(* Logix 5000 project; controller RSL5k_18_Template_noLib Emulate 5570 rev 32.11; software revision 32.02; part 6 of 16 *)
(* tags used below, declared in another part *)
   P_Intlk : BOOL;   // Unique Parameter Name for auto - discovery
(* P_Intlk, continued *)

ROUTINE Prescan   (* ladder *)
// Clear "lurking" Commands
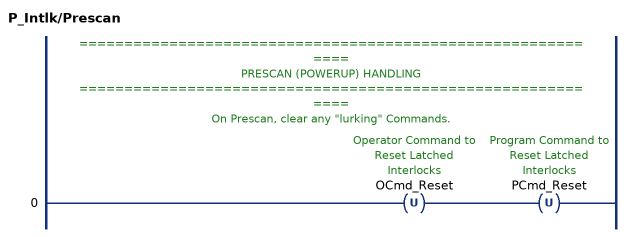
   // ============================================================
   // PRESCAN (POWERUP) HANDLING
   // ============================================================
   // On Prescan, clear any "lurking" Commands.
   0: OTU(OCmd_Reset)OTU(PCmd_Reset);
END_ROUTINE
END_ADD_ON_INSTRUCTION

ADD_ON_INSTRUCTION P_Perm   (* revision 4.10 .00 Release, vendor Rockwell Automation, ExecuteEnableInFalse *)
// Permissives
// Revision note:
// See Instruction Help for a summary of changes, and see 4.10 Release Notes for details.
// Help:
// Copyright © Rockwell Automation, Inc.  All Rights Reserved.
// This Instruction monitors up to 16 Permissive conditions.  It provides these features:
// *  The "OK" state of each Permissive Input is configurable.  By default,
//     each Input is 1 when OK to start, 0 when not OK to start.
// *  Permissives may be configured as Bypassable.  A separate Sts_NBPermOK
//     (Non-Bypassable Permissives OK) status is provided, which the destination
//     object can use for Bypass, Maintenance and other functions,
//     where Bypassable Permissives can be ignored.
// All Permissive Inputs must be in their configured "OK" states
// for the P_Perm instruction to provide a "PermOK" status.
// All non-bypassable Permissive inputs must be in their configured "OK" states
// for the P_Perm instruction to provide a "NBPermOK" status.
// For each Permissive condition, a Tag may be defined for navigation. Clicking
// the Permissive description will call up the associated Tag's Faceplate.
// SUMMARY OF CHANGES FROM PREVIOUS VERSION (4.00.00)
// See 4.10 Release Notes for details.
// * Added Cfg_HasMoreObj.
// SUMMARY OF CHANGES FROM PREVIOUS VERSION (3.5-05)
// See 4.00 Release Notes for details.
// * Changed Inf_ items to HMI_, and added Cfg_Area for security.
// * OSets / OCmds and MSets / MCmds are now LOCAL TAGS.
VAR_INPUT
   Inp_Perm00 : ALIAS FOR Wrk_Inp.0; {visible}   // Permissive Cond 00, OK to start if in configured OK state
   Inp_Perm01 : ALIAS FOR Wrk_Inp.1; {visible}   // Permissive Cond 01, OK to start if in configured OK state
   Inp_Perm02 : ALIAS FOR Wrk_Inp.2; {visible}   // Permissive Cond 02, OK to start if in configured OK state
   Inp_Perm03 : ALIAS FOR Wrk_Inp.3; {visible}   // Permissive Cond 03, OK to start if in configured OK state
   Inp_Perm04 : ALIAS FOR Wrk_Inp.4; {visible}   // Permissive Cond 04, OK to start if in configured OK state
   Inp_Perm05 : ALIAS FOR Wrk_Inp.5; {visible}   // Permissive Cond 05, OK to start if in configured OK state
   Inp_Perm06 : ALIAS FOR Wrk_Inp.6; {visible}   // Permissive Cond 06, OK to start if in configured OK state
   Inp_Perm07 : ALIAS FOR Wrk_Inp.7; {visible}   // Permissive Cond 07, OK to start if in configured OK state
   Inp_Perm08 : ALIAS FOR Wrk_Inp.8;   // Permissive Cond 08, OK to start if in configured OK state
   Inp_Perm09 : ALIAS FOR Wrk_Inp.9;   // Permissive Cond 09, OK to start if in configured OK state
   Inp_Perm10 : ALIAS FOR Wrk_Inp.10;   // Permissive Cond 10, OK to start if in configured OK state
   Inp_Perm11 : ALIAS FOR Wrk_Inp.11;   // Permissive Cond 11, OK to start if in configured OK state
   Inp_Perm12 : ALIAS FOR Wrk_Inp.12;   // Permissive Cond 12, OK to start if in configured OK state
   Inp_Perm13 : ALIAS FOR Wrk_Inp.13;   // Permissive Cond 13, OK to start if in configured OK state
   Inp_Perm14 : ALIAS FOR Wrk_Inp.14;   // Permissive Cond 14, OK to start if in configured OK state
   Inp_Perm15 : ALIAS FOR Wrk_Inp.15;   // Permissive Cond 15, OK to start if in configured OK state
   Inp_BypActive : BOOL; {visible}   // 1=Permissive Bypassing is currently active
   Cfg_OKState : INT := 2#1111_1111_1111_1111;   // Bits indicate which state (0 or 1) of each input is OK to start
   Cfg_Bypassable : INT;   // Set bits indicate which conditions can be bypassed
   Cfg_HasNav : INT;   // Set bits indicate which Navigation buttons are enabled
   Cfg_HasMoreObj : BOOL;   // 1=Tells HMI an object with more info is available
END_VAR
VAR_OUTPUT
   Sts_PermOK : BOOL := 1; {access Read Only, visible}   // Overall Permissive Status (1=OK to start)
   Sts_NBPermOK : BOOL := 1; {access Read Only, visible}   // Non-Bypassable Permissive Status (1 =all non- bypassable Permissives OK to start)
   Sts_BypActive : BOOL; {access Read Only}   // 1=Permissive Bypassing is Active (ignore bypassable permissives)
   Sts_Perm : INT := 2#1111_1111_1111_1111; {access Read Only, visible}   // Individual Permissive Status (1=OK, 0=don't start)
   P_Perm : BOOL;   // Unique Parameter Name for auto - discovery
END_VAR
VAR
   Cfg_CondTxt : STRING_Cond[16] := ([0] := 'Enter Description #0');   // Short HMI description of Permissive Conditions
   Wrk_Inp : INT := 2#1111_1111_1111_1111;   // Collection copy of Inp_PermXXs
   Wrk_Bypass : INT; {access None}   // Working Register for Bypassable Permissives
   HMI_Tab : SINT;   // Tab to display (FTView ME)
   Wrk_InpInv : INT; {access None}   // Input states after inverting based on Cfg_OKState
   HMI_Type : STRING_16 := 'P_Perm'; {access Read Only}   // Type identifier for HMI navigation
   Cfg_Label : STRING_20 := 'Permissives';   // Label for graphic symbol displayed on HMI
   Cfg_Tag : STRING_20 := 'P_Perm';   // Tagname for display on HMI
   Cfg_Desc : STRING_40 := 'Permissives';   // Description for display on HMI
   Cfg_NavTag : STRING_NavTag[16];   // Tagnames for destinations of Navigation buttons
   HMI_Lib : STRING_12 := 'RA-BAS'; {access Read Only}   // Display Library for Faceplate call-up
   MSet_Bypass : INT;   // Individual condition Maintenance Bypass toggles
   Cfg_Area : STRING_Area := 'area01';   // Process Area for security
END_VAR

ROUTINE EnableInFalse   (* ladder *)
// Set summary "OK" Status bits to FALSE (0)
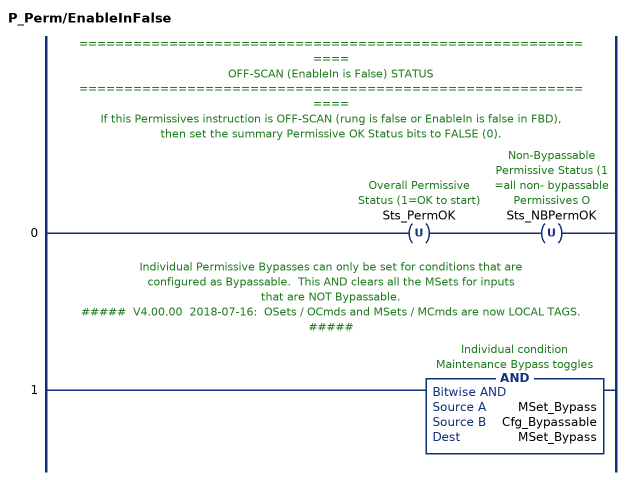
   // ============================================================
   // OFF-SCAN (EnableIn is False) STATUS
   // ============================================================
   // If this Permissives instruction is OFF-SCAN (rung is false or EnableIn is false in FBD),
   // then set the summary Permissive OK Status bits to FALSE (0).
   0: OTU(Sts_PermOK)OTU(Sts_NBPermOK);
   // Individual Permissive Bypasses can only be set for conditions that are
   // configured as Bypassable.  This AND clears all the MSets for inputs
   // that are NOT Bypassable.
   // #####  V4.00.00  2018-07-16:  OSets / OCmds and MSets / MCmds are now LOCAL TAGS.  #####
   1: AND(MSet_Bypass,Cfg_Bypassable,MSet_Bypass);
END_ROUTINE

ROUTINE Logic   (* ladder *)
// Check Permissive Conditions
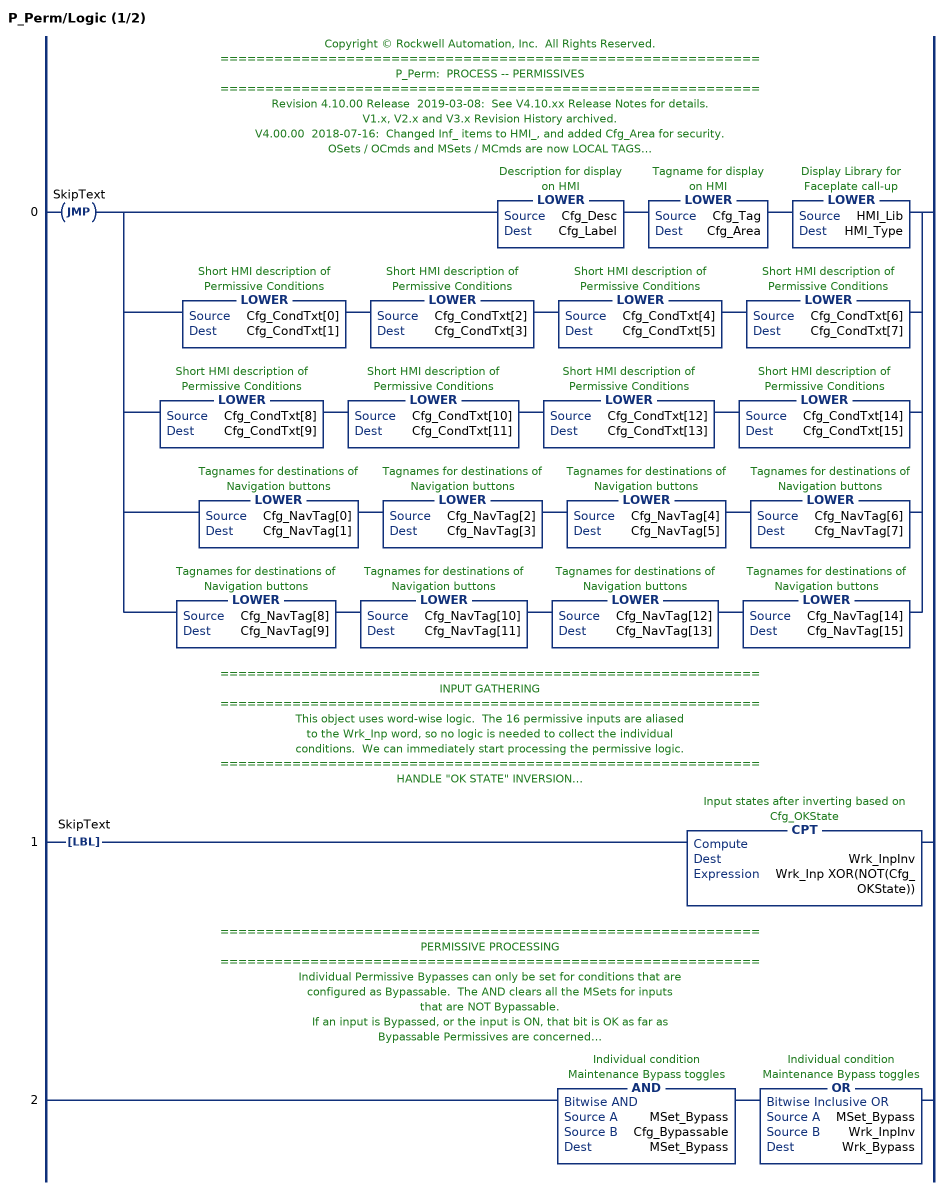
   // Copyright © Rockwell Automation, Inc.  All Rights Reserved.
   // ============================================================
   // P_Perm:  PROCESS -- PERMISSIVES
   // ============================================================
   // Revision 4.10.00 Release  2019-03-08:  See V4.10.xx Release Notes for details.
   // V1.x, V2.x and V3.x Revision History archived.
   // V4.00.00  2018-07-16:  Changed Inf_ items to HMI_, and added Cfg_Area for security.
   // OSets / OCmds and MSets / MCmds are now LOCAL TAGS.
   // V4.10.00  2019-03-08:  Added Cfg_HasMoreObj.
   // ============================================================
   // This Instruction monitors up to 16 Permissive conditions.  It provides these features:
   // *  The "OK" state of each Permissive Input is configurable.  By default,
   // each Input is 1 when OK to start, 0 when not OK to start.
   // *  Permissives may be configured as Bypassable.  A separate Sts_NBPermOK
   // (Non-Bypassable Permissives OK) status is provided, which the destination
   // object can use forBypass, Maintenance and other functions,
   // where Bypassable Permissives can be ignored.
   // All Permissive Inputs must be in their configured "OK" states
   // for the P_Perm instruction to provide a "PermOK" status.
   // All non-bypassable Permissive inputs must be in their configured "OK" states
   // for the P_Perm instruction to provide a "NBPermOK" status.
   // For each Permissive condition, a Tag may be defined for navigation. Clicking
   // the Permissive description will call up the associated Tag's Faceplate.
   // ============================================================
   // SHOW LOCAL STRINGS
   // ============================================================
   // The STRINGs containing the text associated with each instance of this
   // instruction cannot be Input or Output Parameters, because STRINGs are not
   //  'atomic' types. (Inputs and Outputs must be SINT, INT, DINT, REAL, or BOOL.)
   // In order to make it easier to find and configure these STRINGs, this rung
   // was added.  THE JMP (and the LBL on the following rung)
   // MUST NOT BE REMOVED!!!
   // To view the STRINGs, go to the instruction instance (in LD or FBD), RIGHT-click
   // to bring up the context menu and select "Open Instruction Logic".
   // This rung will appear with the STRING values for the selected instance.
   // You may double-click the STRING values here to modify them as well.
   // #####  V4.00.00  2018-07-16:  Added string for Cfg_Area, renamed Inf_* to HMI_*.  #####
   0: JMP(SkipText)[LOWER(Cfg_Desc,Cfg_Label) LOWER(Cfg_Tag,Cfg_Area) LOWER(HMI_Lib,HMI_Type) ,LOWER(Cfg_CondTxt[0],Cfg_CondTxt[1]) LOWER(Cfg_CondTxt[2],Cfg_CondTxt[3]) LOWER(Cfg_CondTxt[4],Cfg_CondTxt[5]) LOWER(Cfg_CondTxt[6],Cfg_CondTxt[7]) ,LOWER(Cfg_CondTxt[8],Cfg_CondTxt[9]) LOWER(Cfg_CondTxt[10],Cfg_CondTxt[11]) LOWER(Cfg_CondTxt[12],Cfg_CondTxt[13]) LOWER(Cfg_CondTxt[14],Cfg_CondTxt[15]) ,LOWER(Cfg_NavTag[0],Cfg_NavTag[1]) LOWER(Cfg_NavTag[2],Cfg_NavTag[3]) LOWER(Cfg_NavTag[4],Cfg_NavTag[5]) LOWER(Cfg_NavTag[6],Cfg_NavTag[7]) ,LOWER(Cfg_NavTag[8],Cfg_NavTag[9]) LOWER(Cfg_NavTag[10],Cfg_NavTag[11]) LOWER(Cfg_NavTag[12],Cfg_NavTag[13]) LOWER(Cfg_NavTag[14],Cfg_NavTag[15]) ];
   // ============================================================
   // INPUT GATHERING
   // ============================================================
   // This object uses word-wise logic.  The 16 permissive inputs are aliased
   // to the Wrk_Inp word, so no logic is needed to collect the individual
   // conditions.  We can immediately start processing the permissive logic.
   // ============================================================
   // HANDLE "OK STATE" INVERSIONS
   // ============================================================
   // This rung inverts the Input bits whose "OK State" is 1 (0 to Run).
   // The resulting Wrk_Inp word is ALL ONES if all permissive inputs are "OK".
   1: LBL(SkipText)CPT(Wrk_InpInv,Wrk_Inp XOR(NOT(Cfg_OKState)));
   // ============================================================
   // PERMISSIVE PROCESSING
   // ============================================================
   // Individual Permissive Bypasses can only be set for conditions that are
   // configured as Bypassable.  The AND clears all the MSets for inputs
   // that are NOT Bypassable.
   // If an input is Bypassed, or the input is ON, that bit is OK as far as
   // Bypassable Permissives are concerned.
   // #####  V4.00.00  2018-07-16:  OSets / OCmds and MSets / MCmds are now LOCAL TAGS.  #####
   2: AND(MSet_Bypass,Cfg_Bypassable,MSet_Bypass)OR(MSet_Bypass,Wrk_InpInv,Wrk_Bypass);
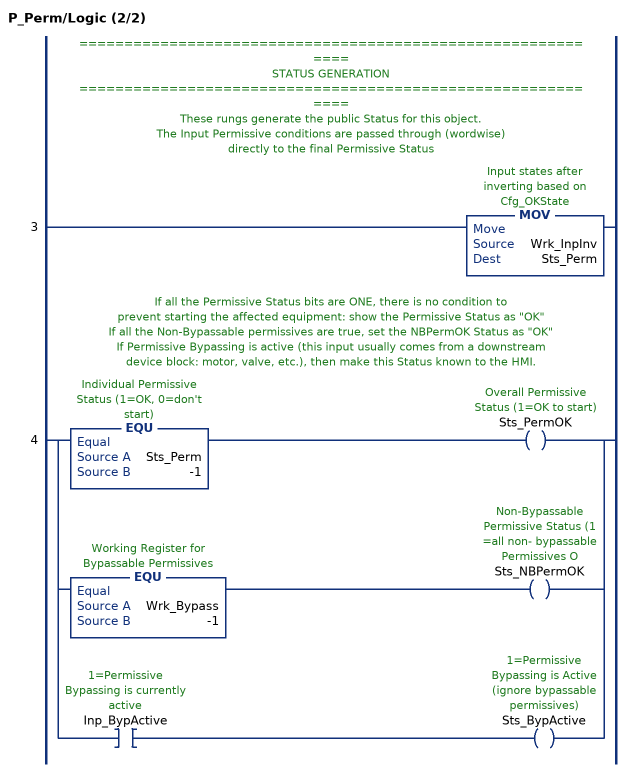
   // ============================================================
   // STATUS GENERATION
   // ============================================================
   // These rungs generate the public Status for this object.
   // The Input Permissive conditions are passed through (wordwise)
   // directly to the final Permissive Status
   3: MOV(Wrk_InpInv,Sts_Perm);
   // If all the Permissive Status bits are ONE, there is no condition to
   // prevent starting the affected equipment: show the Permissive Status as "OK"
   // If all the Non-Bypassable permissives are true, set the NBPermOK Status as "OK"
   // If Permissive Bypassing is active (this input usually comes from a downstream
   // device block: motor, valve, etc.), then make this Status known to the HMI.
   4: [EQU(Sts_Perm,-1) OTE(Sts_PermOK) ,EQU(Wrk_Bypass,-1) OTE(Sts_NBPermOK) ,XIC(Inp_BypActive) OTE(Sts_BypActive) ];
END_ROUTINE
END_ADD_ON_INSTRUCTION

ADD_ON_INSTRUCTION P_PIDE   (* revision 4.10 .01 Release, vendor Rockwell Automation, ExecutePrescan, ExecuteEnableInFalse *)
// Proportional + Integral + Derivative
// Revision note:
// See V4.10.xx Release Notes for details. See Instruction Help for change summary.
// Help:
// Copyright © Rockwell Automation, Inc.  All Rights Reserved.
// This Instruction is used to provide PID (Proportional + Integral +
// Derivative) feedback loop control and provides:
// *  Program and Operator entry of Auto loop mode Setpoint in Engineering Units
// *  Program and Operator entry of Setpoint Target and Ramp Time and
//     command to trigger a Setpoint Ramp ("SP Ramp Wizard")
// *  Program and Operator entry of Manual loop mode Controlled Variable (CV) in Percent
// *  Clamping (in EU) and ramping (in EU/sec) of Setpoint at specified limits
//     (separate increase and decrease rate of change limits).
// *  Clamping (in %) and ramping (in %/sec) of CV at specified limits
//     (separate increase and decrease rate of change limits).
// *  Scaling of Output CV from Percent to CV Engineering Units (CVEU) for use as
//     Cascade Setpoint for a secondary loop or for use as Raw units for an I/O card
// *  Reverse or Direct control action
// *  Feedforward input, feedforward gain, options to add feedforward signal
//     to CV or multiply CV by feedforward signal.
// *  Selection of Velocity (difference) PID form (with inputs for "Previous" CV and FF)
//     or Positional PID form with integral accumulator
// *  Option for fixed bias point positional algorithm in Proportional-only control
//     using Feedforward input to supply bias and with Bumpless transfer,
//     with ramping ("Takeup") rate to return to fixed bias.
// *  Option for Derivative action based on change in Error or change in PV
// *  Option for Proportional action based on Error or PV (Velocity form only)
// *  Monitoring of Interlock conditions which cause output to shed
// *  Configurable shed to HOLD or to configured SAFE value, shed SP to current PV.
// *  Monitoring of I/O communication faults
// *  Alarms for Interlock Trip, Signal Fault, High-High Deviation, High Deviation,
//     Low Deviation and Low-Low Deviation from Setpoint
// *  Operation in Hand, Maintenance, Override, Program and Operator Modes
// *  Full loop control (Cascade, Auto with Setpoint, Manual with CV) available in Override Mode
// *  "Available" status for use by automation logic to know whether loop
//     can be controlled in Auto Mode by other objects.
// SUMMARY OF CHANGES FROM PREVIOUS VERSION (4.10.00)
// See 4.10 Release Notes for details.
// * Corrected clamping of CV, Ratio settings in Manual.
// * Corrected determination of Val_CVSet based on CV Init status.
// * Corrected generation of Sts_PVBad.
// * Modified Interlock function to use PIDE manual CV instead of override CV, to get CV ramping.
// * Corrected SP ramp increasing.
// * Modified Cascade/Ratio logic to include SP rate limiting.
// SUMMARY OF CHANGES FROM PREVIOUS VERSION (4.00.02)
// See 4.10 Release Notes for details.
// * Changed availability to use input availability from interlocks.
// * Corrected parameter and local tag descriptions and external access.
// * Added Cfg_HasMoreObj.
// * Updated to P_CmdSrc V4.10.00.
// * Moved initialization rungs to Logic routine, added Wrk_Init to correct
//     locking of Autotune tag on online instance creation.
// * Corrected overwriting of user SP Rate of Change limits by SP ramp wizard.
// SUMMARY OF CHANGES FROM PREVIOUS VERSION (4.00.01)
// See 4.00 Release Notes for details.
// * Modified handling of CV I/O Fault, CV Fail and Shed configurations.
// * Corrected handling of configured execution interval.
// SUMMARY OF CHANGES FROM PREVIOUS VERSION (4.00.00)
// See 4.00 Release Notes for details.
// * Updated Override Command Source operation and description of
//    Inp_OvrdCmd.
// SUMMARY OF CHANGES FROM PREVIOUS VERSION (3.5-10)
// See 4.00 Release Notes for details.
// * Changed "Mode" to "Command Source", including "External" source.
// * Main Logic routine rewritten in Ladder Diagram.
// * Changed Inf_ items to HMI_, and added Cfg_Area for security.
// * Added notify and unack count rollup for connected objects.
// * Deleted Cfg_PCmdClear.  All Program Commands are now self-clearing.
// * Aligned ready bit naming with command bit names.
// * All OCmds/MCmds and ORdys/MRdys are now Local Tags.
// * Added Sts_RdyAck and Sts_ResetReqd for use by external objects.
// * Added SP Ramping and Ramp Wizard.
// * Added capability to have CV range other than 0 to 100%.
// * Added Shed options.
// * Added Normal Loop Mode, locking of Loop Mode.
// * Added Oper / Prog / Ext "Keep" for Loop Mode, CV, SP, Ratio.
VAR_INPUT
   Inp_PV : ALIAS FOR Wrk_PIDE.PV; {visible}   // Process Variable (PVEU)
   Inp_CascSP : ALIAS FOR Wrk_PIDE.SPCascade; {visible}   // Setpoint in Cascade, Independent PV in Ratio (PVEU)
   Inp_FF : REAL;   // FeedForward term (CVEU)
   Inp_FFPrev : REAL;   // Previous scan FF term (CVEU)
   Inp_CVInitVal : ALIAS FOR Wrk_PIDE.CVInitValue;   // Value to Initialize the CV to when requested (CVRaw)
   Inp_CVPrev : REAL;   // Previous scan CV (CVEU)
   Inp_UseFFPrev : ALIAS FOR Wrk_PIDE.FFSetPrevious;   // 1=Use Inp_FFPrev as previous FF value, 0=Use last scan value
   Inp_UseCVInitVal : ALIAS FOR Wrk_PIDE.CVInitReq;   // 1=Initialize CV to Inp_CVInitValue
   Inp_UseCVPrev : BOOL;   // 1=Use Inp_CVPrev as previous CV value, 0=Use last scan value
   Inp_WindupHi : ALIAS FOR Wrk_PIDE.WindupHIn;   // Windup High Signal, 1=regulator will not increase the integral term
   Inp_WindupLo : ALIAS FOR Wrk_PIDE.WindupLIn;   // Windup Low Signal, 1=regulator will not decrease the integral term
   Inp_PVBad : BOOL;   // 1=PV quality or PV I/O Comms Status Bad, 0=OK
   Inp_PVUncertain : BOOL;   // 1=PV Value Not Reliable, 0=OK
   Inp_CVIOFault : BOOL;   // 1=CV I/O Comms Status Bad, 0=OK
   Inp_PVSrcQ : DINT;   // Source and Quality of Inp_PV (enum)
   Inp_PVNotify : DINT;   // PV Alarm Level and Acknowledgement (enum)
   Inp_CVNotify : DINT;   // CV Alarm Level and Acknowledgement (enum)
   Inp_CascSPNotify : DINT;   // Cascade SP Alarm Level and Acknowledgement (enum)
   Inp_IntlkOK : BOOL := 1; {visible}   // 1=Interlocks OK, CV can be set
   Inp_NBIntlkOK : BOOL := 1; {visible}   // 1=Non-Bypassable Interlocks OK, CV can be set
   Inp_IntlkAvail : BOOL;   // 1 = Interlock Availibility OK
   Inp_Hand : ALIAS FOR CmdSrc.Inp_Hand; {visible}   // 1=Select Hand (hardwired) command source
   Inp_HandFdbk : REAL;   // CV Feedback used in Hand Mode (CVEU)
   Inp_HandFdbkBad : ALIAS FOR Wrk_PIDE.HandFBFault;   // 1=Inp_HandFdbk input quality or I/O Comms Status Bad, 0=OK
   Inp_Ovrd : ALIAS FOR CmdSrc.Inp_Ovrd;   // 1=Select Override command source
   Inp_OvrdCmd : DINT;   // Loop Mode command in Override: 0=None, 1=Man, 2=Auto, 3=Casc, 4=Norm, 5=Start SP Ramp, 6=Stop SP Ramp
   Inp_OvrdRatio : REAL := 1.0;   // Loop Ratio in Override (unitless)
   Inp_OvrdSP : REAL;   // Loop Auto Setpoint (SP) in Override (PVEU)
   Inp_OvrdCV : REAL;   // Loop Manual Output (CV) in Override (CVEU)
   Inp_OvrdSPTarget : REAL;   // Override Setpoint Target for SP Ramping ('wizard') (PVEU)
   Inp_OvrdSPRampT : REAL;   // Override Setpoint Ramp Time for SP Ramping ('wizard') (sec)
   Inp_OvrdSPRoCLimInc : REAL;   // Override Setting for Setpoint Positive Rate of Change Limit (PVEU/sec)
   Inp_OvrdSPRoCLimDec : REAL;   // Override Setting for Setpoint Negative Rate of Change Limit (PVEU/sec)
   Inp_ExtInh : ALIAS FOR CmdSrc.Inp_ExtInh;
   Inp_HiHiDevGate : ALIAS FOR HiHiDevGate.Inp_Gate;   // High-High Deviation Status Gate, 1=enabled
   Inp_HiDevGate : ALIAS FOR HiDevGate.Inp_Gate;   // High Deviation Status Gate, 1=enabled
   Inp_LoDevGate : ALIAS FOR LoDevGate.Inp_Gate;   // Low Deviation Status Gate, 1=enabled
   Inp_LoLoDevGate : ALIAS FOR LoLoDevGate.Inp_Gate;   // Low-Low Deviation Status Gate, 1=enabled
   Inp_Reset : BOOL;   // 1=Reset latched Alarms
   Cfg_HasRatio : ALIAS FOR Wrk_PIDE.UseRatio;   // 1=Casc Loop Mode is Ratio, 0=Casc Loop Mode is Cascade
   Cfg_HasCasc : ALIAS FOR Wrk_PIDE.AllowCasRat;   // 1=Enable the loop to be placed into cascade/ratio mode
   Cfg_HasAuto : BOOL := 1;   // 1=Enable the loop to be placed into automatic mode
   Cfg_HasMan : BOOL := 1;   // 1=Enable the loop to be placed into manual mode
   Cfg_HasSPRamp : BOOL;   // 1=Enable the Setpoint Ramp 'Wizard' function
   Cfg_LockLM : BOOL;   // Lock Loop Mode: 0=not locked, 1=locked in Normal mode (see Cfg_NormLM)
   Cfg_PVTrack : ALIAS FOR Wrk_PIDE.PVTracking;   // 1=SP tracks PV in Manual, 0=no PV tracking
   Cfg_CtrlAction : ALIAS FOR Wrk_PIDE.ControlAction;   // 1=Direct acting (E=PV-SP), 0=Reverse acting (E=SP-PV)
   Cfg_Depend : ALIAS FOR Wrk_PIDE.DependIndepend;   // 1=Dependent gains equation, 0=Independent gains
   Cfg_DerivSmooth : ALIAS FOR Wrk_PIDE.DSmoothing;   // 1=Use Derivative Smoothing
   Cfg_ZCOff : ALIAS FOR Wrk_PIDE.ZCOff;   // 1=need not cross zero error to be in deadband, 0=must cross zero error
   Cfg_PropSPAct : ALIAS FOR Wrk_PIDE.PVEProportional;   // Proportional Action on SP Change 1= None (PV only), 0= Full (Loop Error)
   Cfg_DerivSPAct : ALIAS FOR Wrk_PIDE.PVEDerivative;   // Derivative Action on SP Change 1=None (PV only), 0=Full (Loop Error)
   Cfg_LimitManCV : ALIAS FOR Wrk_PIDE.CVManLimiting;   // 1=CV limits enforced in Manual, 0=No CV Limiting in Manual
   Cfg_InitToMan : ALIAS FOR Wrk_PIDE.ManualAfterInit;   // 1=Go to Manual Loop Mode when an init request is seen
   Cfg_SetTrack : BOOL := 1;   // 1=Prog/Oper/Ext Settings track, 0=no Settings tracking
   Cfg_SetTrackOvrdHand : BOOL;   // 1=Prog/Oper/Ext Settings track Override/Hand Inputs (CV, SP, Ratio)
   Cfg_SkipSPRoCLim : BOOL;   // 1=Skip SP RoC Limiting in Intlk, Maint, Ovrd
   Cfg_HasIntlkObj : BOOL;   // 1=Tells HMI a P_Intlk is connected to Inp_Intlk
   Cfg_HasMoreObj : BOOL;   // 1=Tells HMI an object with more info is available
   Cfg_HasCascSPNav : BOOL;   // 1=Tells HMI to enable navigation to a connected cascade SP object
   Cfg_HasPVNav : BOOL;   // 1=Tells HMI to enable navigation to a connected PV object
   Cfg_HasCVNav : BOOL;   // 1=Tells HMI to enable navigation to a connected CV object
   Cfg_OvrdIntlk : BOOL;   // 1=Override ignores Bypassable Intlk; 0=always use Intlk
   Cfg_IntlkTripLatch : BOOL;   // 1=Latch in Interlock shed action until Reset 0=Return when Interlock clears
   Cfg_SPFailLatch : BOOL;   // 1=Latch in SP Fail shed action until Reset 0=Return when SP is good
   Cfg_PVFailLatch : BOOL;   // 1=Latch in PV Fail shed action until Reset 0=Return when PV is good
   Cfg_CVFailLatch : BOOL;   // 1=Latch in CV Fail shed action until Reset 0=Return when CV is good
   Cfg_NormLM : DINT;   // Normal Loop Mode 0=Disable Normal selection, 1=Man, 2=Auto, 3=Casc
   Cfg_PwrupLM : DINT;   // Powerup Loop Mode 0=No change (last), 1=Man (w/ CV), 2=Auto (w/ SP), 3=Casc, 4=Normal
   Cfg_IntlkTripSPAct : DINT;   // Interlock Trip Setpoint Action: 0=none, 1=hold last good, 2=use Cfg_IntlkSP, 3=set SP to curr. PV
   Cfg_SPFailSPAct : DINT := 1;   // SP Fail Setpoint Action: 1=hold last good, 2=use Cfg_IntlkSP, 3=set SP to curr. PV
   Cfg_PVFailSPAct : DINT;   // PV Fail Setpoint Action: 0=none, 1=hold last good, 2=use Cfg_IntlkSP
   Cfg_CVFailSPAct : DINT;   // CV Fail Setpoint Action: 0=none, 1=hold last good, 2=use Cfg_IntlkSP, 3=set SP to curr. PV
   Cfg_IntlkTripCVAct : DINT := 2;   // Interlock Trip CV Action: 0=none, 1=hold last good, 2=use Cfg_IntlkCV
   Cfg_SPFailCVAct : DINT := 1;   // SP Fail CV Action: 0=none, 1=hold last good, 2=use Cfg_IntlkCV
   Cfg_PVFailCVAct : DINT := 1;   // PV Fail CV Action: 1=hold last good, 2=use Cfg_IntlkCV
   Cfg_CVFailCVAct : DINT := 1;   // CV Fail CV Action: 1=hold last good, 2=use Cfg_IntlkCV
   Cfg_IntlkTripLMAct : DINT;   // Interlock Trip Loop Mode Action: 0=none, 1=Man only, 2=Auto or Man only
   Cfg_SPFailLMAct : DINT;   // SP Fail Loop Mode Action: 0=none, 1=Man only, 2=Auto or Man only
   Cfg_PVFailLMAct : DINT;   // PV Fail Loop Mode Action: 0=none, 1=Man only, 2=Auto or Man only
   Cfg_CVFailLMAct : DINT;   // CV Fail Loop Mode Action: 0=none, 1=Man only, 2=Auto or Man only
   Cfg_PVDecPlcs : DINT := 2;   // Number of decimal places for display of PV / SP
   Cfg_CVDecPlcs : DINT := 2;   // Number of decimal places for display of CV
   Cfg_HasHiHiDevAlm : ALIAS FOR HiHiDev.Cfg_Exists;   // 1=High-High Deviation Alarm exists and will be checked
   Cfg_HasHiDevAlm : ALIAS FOR HiDev.Cfg_Exists;   // 1=High Deviation Alarm exists and will be checked
   Cfg_HasLoDevAlm : ALIAS FOR LoDev.Cfg_Exists;   // 1=Low Deviation Alarm exists and will be checked
   Cfg_HasLoLoDevAlm : ALIAS FOR LoLoDev.Cfg_Exists;   // 1=Low-Low Deviation Alarm exists and will be checked
   Cfg_HasIntlkTripAlm : ALIAS FOR IntlkTrip.Cfg_Exists;   // 1=Interlock Trip Alarm exists and will be checked
   Cfg_HasFailAlm : ALIAS FOR Fail.Cfg_Exists;   // 1=Loop Failure Alarm exists and will be checked
   Cfg_HiHiDevResetReqd : ALIAS FOR HiHiDev.Cfg_ResetReqd;   // 1=Reset required to clear High-High Deviation Alarm
   Cfg_HiDevResetReqd : ALIAS FOR HiDev.Cfg_ResetReqd;   // 1=Reset required to clear High Deviation Alarm
   Cfg_LoDevResetReqd : ALIAS FOR LoDev.Cfg_ResetReqd;   // 1=Reset required to clear Low Deviation Alarm
   Cfg_LoLoDevResetReqd : ALIAS FOR LoLoDev.Cfg_ResetReqd;   // 1=Reset required to clear Low-Low Deviation Alarm
   Cfg_IntlkTripResetReqd : ALIAS FOR IntlkTrip.Cfg_ResetReqd;   // 1=Reset required to clear Interlock Trip Alarm
   Cfg_FailResetReqd : ALIAS FOR Fail.Cfg_ResetReqd;   // 1=Reset required to clear Loop Failure Alarm
   Cfg_HiHiDevAckReqd : ALIAS FOR HiHiDev.Cfg_AckReqd;   // 1=Acknowledge required for High-High Deviation Alarm
   Cfg_HiDevAckReqd : ALIAS FOR HiDev.Cfg_AckReqd;   // 1=Acknowledge required for High Deviation Alarm
   Cfg_LoDevAckReqd : ALIAS FOR LoDev.Cfg_AckReqd;   // 1=Acknowledge required for Low Deviation Alarm
   Cfg_LoLoDevAckReqd : ALIAS FOR LoLoDev.Cfg_AckReqd;   // 1=Acknowledge required for Low-Low Deviation Alarm
   Cfg_IntlkTripAckReqd : ALIAS FOR IntlkTrip.Cfg_AckReqd;   // 1=Acknowledge required for Interlock Trip Alarm
   Cfg_FailAckReqd : ALIAS FOR Fail.Cfg_AckReqd;   // 1=Acknowledge required for Loop Failure Alarm
   Cfg_HiHiDevSeverity : ALIAS FOR HiHiDev.Cfg_Severity;   // High-High Deviation Severity 1..250=Low, 251..500=Medium, 501..750=High, 751..1000=Urgent
   Cfg_HiDevSeverity : ALIAS FOR HiDev.Cfg_Severity;   // High Deviation Severity 1..250=Low, 251..500=Medium, 501..750=High, 751..1000=Urgent
   Cfg_LoDevSeverity : ALIAS FOR LoDev.Cfg_Severity;   // Low Deviation Severity 1..250=Low, 251..500=Medium, 501..750=High, 751..1000=Urgent
   Cfg_LoLoDevSeverity : ALIAS FOR LoLoDev.Cfg_Severity;   // Low-Low Deviation Severity 1..250=Low, 251..500=Medium, 501..750=High, 751..1000=Urgent
   Cfg_IntlkTripSeverity : ALIAS FOR IntlkTrip.Cfg_Severity;   // Interlock Trip Alarm Severity 1..250=Low, 251..500=Medium, 501..750=High, 751..1000=Urgent
   Cfg_FailSeverity : ALIAS FOR Fail.Cfg_Severity;   // Loop Failure Alarm Severity 1..250=Low, 251..500=Medium, 501..750=High, 751..1000=Urgent
   Cfg_MinRatio : ALIAS FOR Wrk_PIDE.RatioLLimit;   // Minimum allowed Ratio (unitless)
   Cfg_MaxRatio : ALIAS FOR Wrk_PIDE.RatioHLimit;   // Maximum allowed Ratio (unitless)
   Cfg_MinSP : ALIAS FOR Wrk_PIDE.SPLLimit;   // Minimum allowed Setpoint (SP) (PVEU)
   Cfg_MaxSP : ALIAS FOR Wrk_PIDE.SPHLimit;   // Maximum allowed Setpoint (SP) (PVEU)
   Cfg_MaxSPRoCInc : REAL;   // Maximum allowed Setpoint Positive Rate of Change Limit (PVEU/sec)
   Cfg_MaxSPRoCDec : REAL;   // Maximum allowed Setpoint Negative Rate of Change Limit (PVEU/sec)
   Cfg_SPRampMaxDev : REAL;   // If deviation exceeds this value, pause SP ramp (0.0=never pause) (PVEU)
   Cfg_PVEUMin : ALIAS FOR Wrk_PIDE.PVEUMin;   // PV Engineering Units Mimimum Value (PVEU)
   Cfg_PVEUMax : ALIAS FOR Wrk_PIDE.PVEUMax;   // PV Engineering Units Maximum Value (PVEU)
   Cfg_CVEUMin : REAL;   // CV Engineering Units Minimum Value (CVEU)
   Cfg_CVEUMax : REAL := 100.0;   // CV Engineering Units Maximum Value (CVEU)
   Cfg_CVRawMin : ALIAS FOR Wrk_PIDE.CVEUMin;   // CV Output Units Minimum Value (CVRaw, for scaling))
   Cfg_CVRawMax : ALIAS FOR Wrk_PIDE.CVEUMax;   // CV Output Units Maximum Value (CVRaw, for scaling)
   Cfg_ExecT : REAL;   // Execution Time (interval) for PID Algorithm (sec)
   Cfg_PGain : ALIAS FOR Wrk_PIDE.PGain;   // Proportional (independent) or Loop (dependent) Gain (unitless)
   Cfg_IGain : ALIAS FOR Wrk_PIDE.IGain;   // Integral Gain (1/min independent or min/repeat dependent)
   Cfg_DGain : ALIAS FOR Wrk_PIDE.DGain;   // Derivative Gain (min)
   Cfg_ZCDB : ALIAS FOR Wrk_PIDE.ZCDeadband;   // Normal Zero Crossing Deadband (PVEU)
   Cfg_MinCV : REAL;   // Minimum allowed Controlled Variable (CV) value (CVEU)
   Cfg_MaxCV : REAL := 100.0;   // Maximum allowed Controlled Variable (CV) value (CVEU)
   Cfg_CVRoCLim : REAL;   // CV Rate of Change Limit (CVEU/sec)
   Cfg_MaxInactiveCV : REAL;   // When Val_CV is greater than this value, set Sts_Active (for HMI) (CVEU)
   Cfg_IntlkSP : REAL;   // SP Value to use with Interlock / Bad Value SP action (PVEU)
   Cfg_IntlkCV : REAL;   // CV Value to use with Interlock / Bad Value CV action (CVEU)
   Cfg_PwrupSP : REAL;   // Loop SP on powerup, used if Cfg_PwrupLM = 1 (Manual) or 2 (Auto) (PVEU)
   Cfg_PwrupCV : REAL;   // Loop CV on powerup, used if Cfg_PwrupLM <> 0 (none) (CVEU)
   Cfg_HiHiDevLim : REAL := 1.5e+38;   // Current High-High Deviation Status Threshold (PVEU)
   Cfg_HiHiDevDB : REAL;   // High-High Devation Status Deadband (PVEU)
   Cfg_HiHiDevOnDly : ALIAS FOR HiHiDevGate.Cfg_OnDly;   // Minimum time above High-High Deviation Limit to raise Status (sec)
   Cfg_HiHiDevOffDly : ALIAS FOR HiHiDevGate.Cfg_OffDly;   // Minimum time below High-High Deviation Limit to clear Status (sec)
   Cfg_HiHiDevGateDly : ALIAS FOR HiHiDevGate.Cfg_GateDly;   // High-High Deviation Status Gate Delay (sec)
   Cfg_HiDevLim : REAL := 1.5e+38;   // Current High Deviation Status Threshold (PVEU)
   Cfg_HiDevDB : REAL;   // High Devation Status Deadband (PVEU)
   Cfg_HiDevOnDly : ALIAS FOR HiDevGate.Cfg_OnDly;   // Minimum time above High Deviation Limit to raise Status (sec)
   Cfg_HiDevOffDly : ALIAS FOR HiDevGate.Cfg_OffDly;   // Minimum time below High Deviation Limit to clear Status (sec)
   Cfg_HiDevGateDly : ALIAS FOR HiDevGate.Cfg_GateDly;   // High Deviation Status Gate Delay (sec)
   Cfg_LoDevLim : REAL := -1.5e+38;   // Current Low Deviation Status Threshold (PVEU)
   Cfg_LoDevDB : REAL;   // Low Devation Status Deadband (PVEU)
   Cfg_LoDevOnDly : ALIAS FOR LoDevGate.Cfg_OnDly;   // Minimum time below Low Deviation Limit to raise Status (sec)
   Cfg_LoDevOffDly : ALIAS FOR LoDevGate.Cfg_OffDly;   // Minimum time above Low Deviation Limit to clear Status (sec)
   Cfg_LoDevGateDly : ALIAS FOR LoDevGate.Cfg_GateDly;   // Low Deviation Status Gate Delay (sec)
   Cfg_LoLoDevLim : REAL := -1.5e+38;   // Current Low-Low Deviation Status Threshold (PVEU)
   Cfg_LoLoDevDB : REAL;   // Low-Low Devation Status Deadband (PVEU)
   Cfg_LoLoDevOnDly : ALIAS FOR LoLoDevGate.Cfg_OnDly;   // Minimum time below Low-Low Deviation Limit to raise Status (sec)
   Cfg_LoLoDevOffDly : ALIAS FOR LoLoDevGate.Cfg_OffDly;   // Minimum time below Low-Low Deviation Limit to clear Status (sec)
   Cfg_LoLoDevGateDly : ALIAS FOR LoLoDevGate.Cfg_GateDly;   // Low-Low Deviation Status Gate Delay (sec)
   Cfg_OperKeep : SINT;   // Oper keeps control: .0=Loop Mode .1=CV .2=SP, .3=Ratio
   Cfg_ProgKeep : SINT;   // Prog keeps control: .0=Loop Mode .1=CV .2=SP, .3=Ratio
   Cfg_ExtKeep : SINT;   // Ext keeps control: .0=Loop Mode .1=CV .2=SP, .3=Ratio
   PSet_Ratio : REAL := 1.0;   // Program Setting for Ratio (loop CasRat and Ratio enabled) (unitless)
   PSet_SP : REAL;   // Program Setting for Setpoint (loop Auto) (PVEU)
   PSet_SPRoCLimInc : REAL;   // Program Setting for Setpoint Rate of Change Limit Increasing (PVEU/sec)
   PSet_SPRoCLimDec : REAL;   // Program Setting for Setpoint Rate of Change Limit Decreasing (PVEU/sec)
   PSet_SPTarget : REAL;   // Program Setting for Setpoint Ramp Target (endpoint, for ramp wizard) (PVEU)
   PSet_SPRampT : REAL;   // Program Setting for Setpoint Ramp Time (to reach target, for ramp wizard) (sec)
   PSet_CV : REAL;   // Program Setting for Controlled Variable (loop Manual) (CVEU)
   PSet_Owner : DINT;   // Program Owner Request ID (non-zero) or Release (zero)
   XSet_Ratio : REAL := 1.0;   // External Setting for Ratio (loop CasRat and Ratio enabled) (unitless)
   XSet_SP : REAL;   // External Setting for Setpoint (loop Auto) (PVEU)
   XSet_SPRoCLimInc : REAL;   // External Setting for Setpoint Rate of Change Limit Increasing (PVEU/sec)
   XSet_SPRoCLimDec : REAL;   // External Setting for Setpoint Rate of Change Limit Decreasing (PVEU/sec)
   XSet_SPTarget : REAL;   // External Setting for Setpoint Ramp Target (endpoint, for ramp wizard) (PVEU)
   XSet_SPRampT : REAL;   // External Setting for Setpoint Ramp Time (to reach target, for ramp wizard) (sec)
   XSet_CV : REAL;   // External Setting for Controlled Variable (loop Manual) (CVEU)
   PCmd_Casc : BOOL;   // Program Command to select Cascade / Ratio Loop Mode
   PCmd_Auto : BOOL;   // Program Command to select Automatic Loop Mode
   PCmd_Man : BOOL;   // Program Command to select Manual Loop Mode
   PCmd_NormLM : BOOL;   // Operator Command to select Normal Loop Mode (see Cfg_NormLM)
   PCmd_SPRampStart : BOOL;   // Program Command to initiate SP ramping
   PCmd_SPRampStop : BOOL;   // Program Command to stop SP ramping
   PCmd_Prog : ALIAS FOR CmdSrc.PCmd_Prog;
   PCmd_Oper : ALIAS FOR CmdSrc.PCmd_Oper;
   PCmd_Lock : ALIAS FOR CmdSrc.PCmd_Lock;
   PCmd_Unlock : ALIAS FOR CmdSrc.PCmd_Unlock;
   PCmd_Normal : ALIAS FOR CmdSrc.PCmd_Normal;
   PCmd_Reset : BOOL;   // Program Command to Reset all Alarms requiring Reset
   PCmd_HiHiDevAck : ALIAS FOR HiHiDev.PCmd_Ack;   // Program Command to Acknowledge High-High Deviation Alarm
   PCmd_HiHiDevSuppress : ALIAS FOR HiHiDev.PCmd_Suppress;   // Program Command to Suppress High-High Deviation Alarm
   PCmd_HiHiDevUnsuppress : ALIAS FOR HiHiDev.PCmd_Unsuppress;   // Program Command to Unsuppress High-High Deviation Alarm
   PCmd_HiHiDevUnshelve : ALIAS FOR HiHiDev.PCmd_Unshelve;   // Program Command to Unshelve High-High Deviation Alarm
   PCmd_HiDevAck : ALIAS FOR HiDev.PCmd_Ack;   // Program Command to Acknowledge High Deviation Alarm
   PCmd_HiDevSuppress : ALIAS FOR HiDev.PCmd_Suppress;   // Program Command to Suppress High Deviation Alarm
   PCmd_HiDevUnsuppress : ALIAS FOR HiDev.PCmd_Unsuppress;   // Program Command to Unsuppress High Deviation Alarm
   PCmd_HiDevUnshelve : ALIAS FOR HiDev.PCmd_Unshelve;   // Program Command to Unshelve High Deviation Alarm
   PCmd_LoDevAck : ALIAS FOR LoDev.PCmd_Ack;   // Program Command to Acknowledge Low Deviation Alarm
   PCmd_LoDevSuppress : ALIAS FOR LoDev.PCmd_Suppress;   // Program Command to Suppress Low Deviation Alarm
   PCmd_LoDevUnsuppress : ALIAS FOR LoDev.PCmd_Unsuppress;   // Program Command to Unsuppress Low Deviation Alarm
   PCmd_LoDevUnshelve : ALIAS FOR LoDev.PCmd_Unshelve;   // Program Command to Unshelve Low Deviation Alarm
   PCmd_LoLoDevAck : ALIAS FOR LoLoDev.PCmd_Ack;   // Program Command to Acknowledge Low-Low Deviation Alarm
   PCmd_LoLoDevSuppress : ALIAS FOR LoLoDev.PCmd_Suppress;   // Program Command to Suppress Low-Low Deviation Alarm
   PCmd_LoLoDevUnsuppress : ALIAS FOR LoLoDev.PCmd_Unsuppress;   // Program Command to Unsuppress Low-Low Deviation Alarm
   PCmd_LoLoDevUnshelve : ALIAS FOR LoLoDev.PCmd_Unshelve;   // Program Command to Unshelve Low-Low Deviation Alarm
   PCmd_IntlkTripAck : ALIAS FOR IntlkTrip.PCmd_Ack;   // Program Command to Acknowledge Interlock Trip Alarm
   PCmd_IntlkTripSuppress : ALIAS FOR IntlkTrip.PCmd_Suppress;   // Program Command to Suppress Interlock Trip Alarm
   PCmd_IntlkTripUnsuppress : ALIAS FOR IntlkTrip.PCmd_Unsuppress;   // Program Command to Unsuppress Interlock Trip Alarm
   PCmd_IntlkTripUnshelve : ALIAS FOR IntlkTrip.PCmd_Unshelve;   // Program Command to Unshelve Interlock Trip Alarm
   PCmd_FailAck : ALIAS FOR Fail.PCmd_Ack;   // Program Command to Acknowledge Loop Failure Alarm
   PCmd_FailSuppress : ALIAS FOR Fail.PCmd_Suppress;   // Program Command to Suppress Loop Failure Alarm
   PCmd_FailUnsuppress : ALIAS FOR Fail.PCmd_Unsuppress;   // Program Command to Unsuppress Loop Failure Alarm
   PCmd_FailUnshelve : ALIAS FOR Fail.PCmd_Unshelve;   // Program Command to Unshelve Loop Failure Alarm
   MCmd_Rel : ALIAS FOR CmdSrc.MCmd_Rel;
   OCmd_Unlock : ALIAS FOR CmdSrc.OCmd_Unlock;
   XCmd_Casc : BOOL;   // External Command to select Cascade / Ratio control
   XCmd_Auto : BOOL;   // External Command to select Automatic control
   XCmd_Man : BOOL;   // External Command to select Manual control
   XCmd_NormLM : BOOL;   // External Command to select Normal Loop Mode (see Cfg_NormLM)
   XCmd_SPRampStart : BOOL;   // External Command to initiate SP ramping
   XCmd_SPRampStop : BOOL;   // External Command to stop SP ramping
   XCmd_Acq : ALIAS FOR CmdSrc.XCmd_Acq;
   XCmd_Rel : ALIAS FOR CmdSrc.XCmd_Rel;
   XCmd_Reset : BOOL;   // External Command to Reset all Alarms requiring Reset
END_VAR
VAR_OUTPUT
   Out_CV : ALIAS FOR Wrk_PIDE.CVEU; {visible}   // CV to final control element (CV Raw Units)
   Val_PV : REAL; {access Read Only, visible}   // Value of Loop PV (PVEU)
   Val_Ratio : ALIAS FOR Wrk_PIDE.Ratio;   // Value of Loop Ratio (unitless)
   Val_SPSet : REAL; {access Read Only}   // Value of selected SP (before clamping and ramping) (PVEU)
   Val_SP : ALIAS FOR Wrk_PIDE.SP; {visible}   // Value of SP being used (after ramping and clamping (PVEU)
   Val_SPTarget : REAL; {access Read Only}   // Accepted Setting for Setpoint Ramp Target (endpoint, for ramp wizard) (PVEU)
   Val_SPRampT : REAL; {access Read Only}   // Accepted Setting for Setpoint Ramp Time (to reach target, for ramp wizard) (sec)
   Val_SPRampRoC : REAL; {access Read Only}   // Calculated Value of SP Rate of Change for Ramping (from Ramp Wizard) (PVEU/sec)
   Val_SPRoCInc : REAL; {access Read Only}   // Current Value of Setpoint Rate of Change Limit Increasing (PVEU/sec)
   Val_SPRoCDec : REAL; {access Read Only}   // Current Value of Setpoint Rate of Change Limit Decreasing (PVEU/sec)
   Val_E : ALIAS FOR Wrk_PIDE.E;   // Loop Error (PV-SP) (PVEU)
   Val_CVSet : REAL; {access Read Only, visible}   // Value of selected CV (before clamping and ramping) (CVEU)
   Val_CVOut : REAL; {access Read Only, visible}   // Value of CV Output (after ramping and clamping (CVEU)
   Val_PVPercent : ALIAS FOR Wrk_PIDE.PVPercent;   // Loop PV (percent of span)
   Val_SPPercent : ALIAS FOR Wrk_PIDE.SPPercent;   // Loop SP (percent of span)
   Val_EPercent : ALIAS FOR Wrk_PIDE.EPercent;   // Loop Error (PV-SP) (percent of span)
   Val_CVPercent : ALIAS FOR Wrk_PIDE.CV;   // Loop CV (percent of span)
   Val_ActExecT : ALIAS FOR Wrk_PIDE.DeltaT;   // Actual PID Algorithm Execution Time (Interval) (sec)
   Val_Init : REAL; {access Read Only}   // Initialization Value for this loop's Cascade Primary (PVEU)
   Val_PVEUMin : REAL; {access Read Only}   // Minimum of PV scaled range (PVEU)
   Val_PVEUMax : REAL := 100.0; {access Read Only}   // Maximum of PV scaled range (PVEU)
   Val_CVEUMin : REAL; {access Read Only}   // Minimum of CV scaled range (CVEU)
   Val_CVEUMax : REAL := 100.0; {access Read Only}   // Maximum of CV scaled range (CVEU)
   SrcQ_IO : DINT; {access Read Only}   // Source and Quality of primary I/O (enumeration)
   SrcQ : DINT; {access Read Only}   // Source and Quality of primary Val/Sts (enumeration)
   Val_Sts : DINT; {access Read Only}   // Loop Status enum: 0=unknown (POoS @ Intlk CV), 1=Manual, 2=Auto, 3=Cascade (no ratio), 4=Ratio
   Val_Fault : DINT; {access Read Only}   // Loop Fault: 0=none, 1=PV Uncertain, 22=LoDev, 23=HiDev, 27=LLDev, 28=HHDev, 29=Intlk Trip, 30=SP Fail, 31=PV Fail, 32=CV Fail, 34=Cfg Err
   Val_State : DINT; {access Read Only}   // Loop State: 0=Man, 1=In DB, 2=Not in DB, 3=SPRamp, 4=CVRamp, 5=Ratio Clamp, 6=SP Clamp, 7=CV Clamp, 8=Windup L, 9=Windup H, 10=SP Held, 11=SP @ IntlkSP, 12 = CV Held, 13=CV @ Intlk CV, 14=Hand, 15=Init
   Val_NotifyAll : DINT; {access Read Only}   // Highest Alarm prio and ack status this object + PV, CV, CascSP (enum)
   Val_UnackAlmC : DINT; {access Read Only}   // Count of Unacknowledged Alarms
   Val_Owner : DINT; {access Read Only}   // Current Object Owner ID (0=not owned)
   Sts_InstrFaults1 : DINT; {access Read Only}   // PIDE Block Status1 Instruction Fault bits (See PIDE Instruction Help)
   Sts_InstrFaults2 : DINT; {access Read Only}   // PIDE Block Status2 Instruction Fault bits (See PIDE Instruction Help)
   Sts_Casc : BOOL; {access Read Only, visible}   // 1=Loop Mode is Cascade/Ratio
   Sts_Auto : BOOL; {access Read Only, visible}   // 1=Loop Mode is Auto
   Sts_Man : BOOL; {access Read Only, visible}   // 1=Loop Mode is Manual
   Sts_NormLM : BOOL; {access Read Only}   // 1=Loop is in Normal Loop Mode (see Cfg_NormLM)
   Sts_Initializing : ALIAS FOR Wrk_PIDE.CVInitializing;   // 1=CV is initializing because of Request from this loop's Secondary
   Sts_InitReq : BOOL;   // 1=CV Initialize Request to this loop's Primary
   Sts_WindupHi : ALIAS FOR Wrk_PIDE.WindupHOut;   // 1=This loop winding up High, to Inp_WindupHi of this loop's Primary
   Sts_WindupLo : ALIAS FOR Wrk_PIDE.WindupLOut;   // 1=This loop winding up Low, to Inp_WindupLo of this loop's Primary
   Sts_ZCDBOn : ALIAS FOR Wrk_PIDE.ZCDeadbandOn;   // Deadband Indicator: 1=PV is within ZC deadband and CV will not change
   Sts_RatioClamped : BOOL; {access Read Only}   // 1=Selected Ratio (PSet/OSet_Ratio or Inp_OvrdRatio) has been clamped
   Sts_SPBad : ALIAS FOR Wrk_PIDE.SPProgInv;   // 1=SP Value is Bad (quality) or invalid or Casc SP comms fault
   Sts_IntlkSP : BOOL; {access Read Only}   // 1=SP Value is being set by shed to Interlock SP
   Sts_SPHeld : BOOL; {access Read Only}   // 1=SP Value is being set by shed to hold last good SP
   Sts_SPShedPV : BOOL; {access Read Only}   // 1=SP Value was set by shed to current PV
   Sts_SPShed : BOOL; {access Read Only}   // 1=SP from Shed, 0=SP from Prog, Oper, Ovrd (A), Casc SP Input (C) or PV Track (M)
   Sts_SPTrackPV : BOOL; {access Read Only}   // 1=SP Value is being set by PV Tracking (in Manual Mode)
   Sts_SPClamped : BOOL; {access Read Only}   // 1=Selected SP is being clamped (for faceplate animation)
   Sts_SPRamping : BOOL; {access Read Only}   // 1=SP is ramping toward Val_SPSet, 0=ramp complete
   Sts_SkipSPRoCLim : BOOL; {access Read Only}   // 1=SP rate limiting is being skipped (for faceplate animation)
   Sts_PVBad : BOOL; {access Read Only}   // 1=PV Value, comms, quality or EU Limitis Bad
   Sts_PVUncertain : BOOL; {access Read Only}   // 1=PV Value is Uncertain (quality)
   Sts_FFBad : ALIAS FOR Wrk_PIDE.FFInv;   // 1=Feedforward Term Value is invalid
   Sts_FFPrevBad : ALIAS FOR Wrk_PIDE.FFPreviousInv;   // 1=Inp_FFPrev is <-100 CV%, >100 CV%, or not a number (NaN)
   Sts_CVBad : BOOL; {access Read Only}   // 1=CV Value is Bad (quality) or invalid or CV comms fault
   Sts_CVPrevBad : ALIAS FOR Wrk_PIDE.CVPreviousInv;   // 1=Inp_CVPrev is <0.0 CV%, >100.0 CV%, or not a number (NaN)
   Sts_HandFdbkBad : ALIAS FOR Wrk_PIDE.HandFBFaulted;   // 1=Hand FB (Tieback) Value is Bad (quality) or invalid or comms fault
   Sts_IntlkCV : BOOL; {access Read Only}   // 1=CV Value is being set by shed to Interlock CV
   Sts_CVHeld : BOOL; {access Read Only}   // 1=CV Value is being set by shed to hold last good CV
   Sts_CVShed : BOOL; {access Read Only}   // 1=CV from Shed, 0=CV from Prog, Oper, Ovrd (Man), or PID (Auto, Casc)
   Sts_CVClamped : BOOL; {access Read Only}   // 1=Selected CV is being clamped (for faceplate animation)
   Sts_CVRamping : ALIAS FOR Wrk_PIDE.CVROCAlarm;   // 1=CV is ramping toward Val_CVSet, 0=ramp complete
   Sts_Active : BOOL; {access Read Only}   // 1=CV is greater than Cfg_MaxInactiveCV, show graphic symbol as "active"
   Sts_Available : BOOL; {access Read Only}   // 1=PID Loop is available for control by automation (Prog)
   Sts_Bypass : BOOL; {access Read Only}   // 1=Bypassable Interlocks are Bypassed
   Sts_BypActive : BOOL; {access Read Only}   // 1=Bypassing Active (Bypassed or Maintenance)
   Sts_NotRdy : BOOL; {access Read Only}   // 1=Device Not Ready, see detail bits for reason
   Nrdy_CfgErr : BOOL; {access Read Only}   // 1=Device Not Ready: Configuration Error
   Nrdy_Init : BOOL; {access Read Only}   // 1=Device Not Ready: Initialized to Manual Mode
   Nrdy_Intlk : BOOL; {access Read Only}   // 1=Device Not Ready: Interlock Not OK
   Nrdy_IOFault : BOOL; {access Read Only}   // 1=Device Not Ready: I/O Fault (Shed Requires Reset)
   Nrdy_OoS : BOOL; {access Read Only}   // 1=Device Not Ready: Out of Service
   Sts_MaintByp : BOOL; {access Read Only}   // 1=Device has a Maintenance Bypass function active
   Sts_AlmInh : BOOL; {access Read Only}   // 1=One or more Alarms Shelved, Disabled or Suppressed
   Sts_Err : BOOL; {access Read Only, visible}   // 1=Error in Config: see detail Err bits for reason
   Err_Timer : BOOL; {access Read Only}   // 1=Error in Config: Status On-Delay or Off-Delay Time Invalid
   Err_Alarm : BOOL; {access Read Only}   // 1=Error in Config: Alarm Severity Invalid
   Err_RatioLim : ALIAS FOR Wrk_PIDE.RatioLimitsInv;   // 1=Error in Config: Ratio Clamping Limits Invalid
   Err_SPLim : ALIAS FOR Wrk_PIDE.SPLimitsInv;   // 1=Error in Config: Setpoint Clamping Limits Invalid
   Err_CVLim : ALIAS FOR Wrk_PIDE.CVLimitsInv;   // 1=Error in Config: CV Clamping Limits Invalid
   Err_PVEU : ALIAS FOR Wrk_PIDE.PVSpanInv;   // 1=Error in Config: PV EU Max/Min Invalid
   Err_CVEU : BOOL; {access Read Only}   // 1=Error in Config: CV EU Max/Min Invalid
   Err_CVRaw : ALIAS FOR Wrk_PIDE.CVEUSpanInv;   // 1=Error in Config: CV Raw Max/Min Invalid
   Err_ZCDB : ALIAS FOR Wrk_PIDE.ZCDeadbandInv;   // 1=Error in Config: Loop Zero Crossing Deadband Invalid
   Sts_Hand : ALIAS FOR CmdSrc.Sts_Hand; {access Read Only, visible}
   Sts_OoS : ALIAS FOR CmdSrc.Sts_OoS; {access Read Only, visible}
   Sts_Maint : ALIAS FOR CmdSrc.Sts_Maint; {access Read Only, visible}
   Sts_Ovrd : ALIAS FOR CmdSrc.Sts_Ovrd; {access Read Only, visible}
   Sts_Ext : ALIAS FOR CmdSrc.Sts_Ext; {access Read Only, visible}
   Sts_Prog : ALIAS FOR CmdSrc.Sts_Prog; {access Read Only, visible}
   Sts_ProgLocked : ALIAS FOR CmdSrc.Sts_ProgLocked; {access Read Only}
   Sts_Oper : ALIAS FOR CmdSrc.Sts_Oper; {access Read Only, visible}
   Sts_OperLocked : ALIAS FOR CmdSrc.Sts_OperLocked; {access Read Only}
   Sts_Normal : ALIAS FOR CmdSrc.Sts_Normal; {access Read Only}
   Sts_ExtReqInh : ALIAS FOR CmdSrc.Sts_ExtReqInh; {access Read Only}
   Sts_ProgReqInh : ALIAS FOR CmdSrc.Sts_ProgReqInh; {access Read Only}
   Sts_MAcqRcvd : ALIAS FOR CmdSrc.Sts_MAcqRcvd; {access Read Only}
   Sts_RdyReset : ALIAS FOR ORdy_Reset; {access Read Only}   // 1=A latched alarm or shed condition is ready to be reset
   Sts_RdyAck : BOOL; {access Read Only}   // 1=An alarm is ready to be acknowledged
   Sts_HiHiDevCmp : ALIAS FOR HiHiDevGate.Inp;   // High-High Deviation comparison result 1=High-High
   Sts_HiHiDevGate : ALIAS FOR HiHiDevGate.Sts_Gate; {access Read Only}   // High-High Deviation Gate Delay Status, 1=done
   Sts_HiHiDev : ALIAS FOR HiHiDev.Inp;   // 1=PV Deviation is above High-High limit
   Alm_HiHiDev : ALIAS FOR HiHiDev.Alm;   // 1=Loop High-High Deviation Alarm
   Ack_HiHiDev : ALIAS FOR HiHiDev.Ack;   // 1=High-High Deviation Alarm has been acknowledged
   Sts_HiHiDevDisabled : ALIAS FOR HiHiDev.Disabled;   // 1=High-High Deviation Alarm is Disabled (by Maint)
   Sts_HiHiDevShelved : ALIAS FOR HiHiDev.Shelved;   // 1=High-High Deviation Alarm is Shelved (by Oper)
   Sts_HiHiDevSuppressed : ALIAS FOR HiHiDev.Suppressed;   // 1=High-High Deviation Alarm is Suppressed (by logic)
   Sts_HiDevCmp : ALIAS FOR HiDevGate.Inp;   // High Deviation comparison result 1=High-High
   Sts_HiDevGate : ALIAS FOR HiDevGate.Sts_Gate; {access Read Only}   // High Deviation Gate Delay Status, 1=done
   Sts_HiDev : ALIAS FOR HiDev.Inp;   // 1=PV Deviation is above High limit
   Alm_HiDev : ALIAS FOR HiDev.Alm;   // 1=Loop High Deviation Alarm
   Ack_HiDev : ALIAS FOR HiDev.Ack;   // 1=High Deviation Alarm has been acknowledged
   Sts_HiDevDisabled : ALIAS FOR HiDev.Disabled;   // 1=High Deviation Alarm is Disabled (by Maint)
   Sts_HiDevShelved : ALIAS FOR HiDev.Shelved;   // 1=High Deviation Alarm is Shelved (by Oper)
   Sts_HiDevSuppressed : ALIAS FOR HiDev.Suppressed;   // 1=High Deviation Alarm is Suppressed (by logic)
   Sts_LoDevCmp : ALIAS FOR LoDevGate.Inp;   // Low Deviation comparison result 1=High-High
   Sts_LoDevGate : ALIAS FOR LoDevGate.Sts_Gate; {access Read Only}   // Low Deviation Gate Delay Status, 1=done
   Sts_LoDev : ALIAS FOR LoDev.Inp;   // 1=PV Deviation is below Low limit
   Alm_LoDev : ALIAS FOR LoDev.Alm;   // 1=Loop Low Deviation Alarm
   Ack_LoDev : ALIAS FOR LoDev.Ack;   // 1=Loiw Deviation Alarm has been acknowledged
   Sts_LoDevDisabled : ALIAS FOR LoDev.Disabled;   // 1=Low Deviation Alarm is Disabled (by Maint)
   Sts_LoDevShelved : ALIAS FOR LoDev.Shelved;   // 1=Low Deviation Alarm is Shelved (by Oper)
   Sts_LoDevSuppressed : ALIAS FOR LoDev.Suppressed;   // 1=Low Deviation Alarm is Suppressed (by logic)
   Sts_LoLoDevCmp : ALIAS FOR LoLoDevGate.Inp;   // Low-Low Deviation comparison result 1=High-High
   Sts_LoLoDevGate : ALIAS FOR LoLoDevGate.Sts_Gate; {access Read Only}   // Low-Low Deviation Gate Delay Status, 1=done
   Sts_LoLoDev : ALIAS FOR LoLoDev.Inp;   // 1=PV Deviation is below Low-Low limit
   Alm_LoLoDev : ALIAS FOR LoLoDev.Alm;   // 1=Loop Low-Low Deviation Alarm
   Ack_LoLoDev : ALIAS FOR LoLoDev.Ack;   // 1=Low-Loiw Deviation Alarm has been acknowledged
   Sts_LoLoDevDisabled : ALIAS FOR LoLoDev.Disabled;   // 1=Low-Low Deviation Alarm is Disabled (by Maint)
   Sts_LoLoDevShelved : ALIAS FOR LoLoDev.Shelved;   // 1=Low-Low Deviation Alarm is Shelved (by Oper)
   Sts_LoLoDevSuppressed : ALIAS FOR LoLoDev.Suppressed;   // 1=Low-Low Deviation Alarm is Suppressed (by logic)
   Sts_IntlkTrip : ALIAS FOR IntlkTrip.Inp;   // 1=Interlock NOT OK caused loop output to hold or change
   Alm_IntlkTrip : ALIAS FOR IntlkTrip.Alm;   // 1=Interlock Trip Alarm
   Ack_IntlkTrip : ALIAS FOR IntlkTrip.Ack;   // 1=Interlock Trip Alarm has been acknowledged
   Sts_IntlkTripDisabled : ALIAS FOR IntlkTrip.Disabled;   // 1=Interlock Trip Alarm is Disabled (by Maint)
   Sts_IntlkTripShelved : ALIAS FOR IntlkTrip.Shelved;   // 1=Interlock Trip Alarm is Shelved (by Oper)
   Sts_IntlkTripSuppressed : ALIAS FOR IntlkTrip.Suppressed;   // 1=Interlock Trip Alarm is Suppressed (by logic)
   Sts_Fail : ALIAS FOR Fail.Inp;   // 1=Loop Failure: PV Bad, SP Bad or CV Comm Failure or Bad
   Alm_Fail : ALIAS FOR Fail.Alm;   // 1=Loop Failure Alarm: PV Bad, SP Bad or CV Comm Failure or Bad
   Ack_Fail : ALIAS FOR Fail.Ack;   // 1=Loop Failure Alarm has been acknowledged
   Sts_FailDisabled : ALIAS FOR Fail.Disabled;   // 1=Loop Failure Alarm is Disabled (by Maint)
   Sts_FailShelved : ALIAS FOR Fail.Shelved;   // 1=Loop Failure Alarm is Shelved (by Oper)
   Sts_FailSuppressed : ALIAS FOR Fail.Suppressed;   // 1=Loop Failure Alarm is Suppressed (by logic)
   MRdy_Rel : ALIAS FOR CmdSrc.MRdy_Rel; {access Read Only}
   ORdy_Unlock : ALIAS FOR CmdSrc.ORdy_Unlock; {access Read Only}
   P_PIDE : BOOL;   // Unique Parameter Name for auto - discovery
END_VAR
VAR
   CmdSrc : P_CmdSrc := (Cfg_HasOper := 1, Cfg_HasOperLocked := 1, Cfg_HasProg := 1, Cfg_HasProgLocked := 1, Cfg_HasMaint := 1, Cfg_HasMOoS := 1, Cfg_OvrdOverLock := 1, Sts_bSrc := 1);   // Control / Command Source Selection
   Fail : P_Alarm := (Inp := 1, Cfg_AckReqd := 1, Cfg_AllowShelve := 1, Cfg_AllowDisable := 1, Cfg_Severity := 1000, Cfg_AlmMinOnT := 5, PCfg_AllowExist := 1, Ack := 1);   // Loop (SP, PV or CV) Failure Alarm
   IntlkTrip : P_Alarm := (Inp := 1, Cfg_AckReqd := 1, Cfg_AllowShelve := 1, Cfg_AllowDisable := 1, Cfg_Severity := 500, Cfg_AlmMinOnT := 5, PCfg_AllowExist := 1, Ack := 1);   // Interlock Trip Alarm
   Cfg_Tag : STRING_20 := 'P_PIDAdv';   // Tagname displayed on HMI
   Cfg_Label : STRING_20 := 'PID Loop';   // Label for graphic symbol displayed on HMI
   Cfg_Desc : STRING_40 := 'Advanced PID Control Loop';   // Description displayed on HMI
   Wrk_Notify : DINT; {access None}   // Buffer for building Val_Notify
   Wrk_Bypass : BOOL; {access None}   // Internal Bypassable Interlocks are Bypassed flag
   Cfg_PVEU : STRING_8 := '%';   // PV / Setpoint Engineering Units displayed on HMI
   Wrk_ScanTime : REAL; {access None}   // Time since previous scan (sec)
   Wrk_SPStepInc : REAL; {access None}   // Amount to add this scan for SP RoC increasing limiting (PVEU)
   Wrk_ScanT : TIMER := (PRE := 2147483647); {access None}   // Scan Timer (milliseconds, always runs)
   HMI_Tab : SINT;   // Tab to display (FTView ME)
   Wrk_ProgKeepONS : SINT; {access None}   // Program Keep one-shot stores
   Wrk_OperKeepONS : SINT; {access None}   // Operator Keep one-shot stores
   Wrk_ExtKeepONS : SINT; {access None}   // External Keep one-shot stores
   Wrk_State : DINT; {access None}   // Buffer for building Val_State
   Wrk_Sts : DINT; {access None}   // Buffer for building Val_Sts
   Wrk_Fault : DINT; {access None}   // Buffer for building Val_Fault
   LoLoDev : P_Alarm := (Inp := 1, Cfg_AckReqd := 1, Cfg_AllowShelve := 1, Cfg_AllowDisable := 1, Cfg_Severity := 750, Cfg_AlmMinOnT := 5, PCfg_AllowExist := 1, Ack := 1);   // Low-Low Deviation Alarm
   LoDev : P_Alarm := (Inp := 1, Cfg_AckReqd := 1, Cfg_AllowShelve := 1, Cfg_AllowDisable := 1, Cfg_Severity := 500, Cfg_AlmMinOnT := 5, PCfg_AllowExist := 1, Ack := 1);   // Low Deviation Alarm
   HiDev : P_Alarm := (Inp := 1, Cfg_AckReqd := 1, Cfg_AllowShelve := 1, Cfg_AllowDisable := 1, Cfg_Severity := 500, Cfg_AlmMinOnT := 5, PCfg_AllowExist := 1, Ack := 1);   // High Deviation Alarm
   HiHiDev : P_Alarm := (Inp := 1, Cfg_AckReqd := 1, Cfg_AllowShelve := 1, Cfg_AllowDisable := 1, Cfg_Severity := 750, Cfg_AlmMinOnT := 5, PCfg_AllowExist := 1, Ack := 1);   // High-High Deviation Alarm
   Cfg_CVEU : STRING_8 := '%';   // CV Engineering Units displayed on HMI
   Wrk_Casc : BOOL; {access None}   // Internal Loop Mode latch: Cascade selected
   Wrk_Auto : BOOL; {access None}   // Internal Loop Mode latch: 1=Auto selected
   Wrk_Man : BOOL := 1; {access None}   // Internal Loop Mode latch: Manual selected
   Wrk_SPStepDec : REAL; {access None}   // Amount to add this scan for SP RoC decreasing limiting (PVEU)
   Wrk_IntlkOK : BOOL; {access None}   // 1=Interlocks are OK, accounting for bypassing
   HMI_Type : STRING_16 := 'P_PIDE'; {access Read Only}   // Must contain AOI name, used for HMI and Information S/W
   Wrk_IntlkTripShed : BOOL; {access None}   // Shed Latch for Interlock Not OK
   Wrk_PVFailShed : BOOL; {access None}   // Shed Latch for PV Failure
   Wrk_SPFailShed : BOOL; {access None}   // Shed Latch for SP Failure
   Wrk_CVFailShed : BOOL; {access None}   // Shed Latch for CV Failure
   Wrk_AlgoScanT : REAL; {access None}   // Time since last calculation of PID Algorithm (sec)
   Wrk_ShedMan : BOOL; {access None}   // A shed condition is forcing Loop Mode to Manual
   Wrk_ShedAuto : BOOL; {access None}   // A shed condition is forcing Loop Mode to Auto or Manual
   Wrk_SkippedPID : BOOL; {access None}   // PID Algorithm was NOT scanned this time through
   LoLoDevGate : P_Gate := (Inp_Gate := 1);   // Low-Low Deviation Gate/Delay
   LoDevGate : P_Gate := (Inp_Gate := 1);   // Low Deviation Gate/Delay
   HiDevGate : P_Gate := (Inp_Gate := 1);   // High Deviation Gate/Delay
   HiHiDevGate : P_Gate := (Inp_Gate := 1);   // High-High Deviation Gate/Delay
   Val_Notify : DINT; {access Read Only}   // Current Alarm Level and Acknowledgement (enumeration)
   Wrk_SrcQ : DINT; {access None}   // Buffer for building Source / Quality enumeration
   Cfg_CVNavTag : STRING_NavTag;   // Tagname for destination of CV Navigation button
   Cfg_PVNavTag : STRING_NavTag;   // Tagname for destination of PV Navigation button
   Cfg_CascSPNavTag : STRING_NavTag;   // Tagname for destination of Cascade SP Navigation button
   HMI_Lib : STRING_12 := 'RA-BAS'; {access Read Only}   // Display Library for Faceplate call-up
   Wrk_PIDE : PID_ENHANCED := (PVEUMax := 100.0, SPHLimit := 100.0, RatioProg := 1.0, RatioOper := 1.0, RatioHLimit := 1.0, RatioLLimit := 1.0, CVEUMax := 100.0, CVHLimit := 100.0, PVEDerivative := 1, RTSTime := 1, Ratio := 1.0);   // Built-in controller PID algorithm
   Wrk_UnackAlmC : DINT; {access None}   // Buffer for building Val_UnackAlmC
   Cfg_Area : STRING_Area := 'area01';   // Process Area for security
   Wrk_Autotune : PIDE_AUTOTUNE;   // Autotune tag associated with built-in PID algorithm
   Wrk_PIDE_only : P_PIDE_only; {access None}   // Backing tag for AOI containing PIDE (with optional autotune)
   HMI_HasAutotune : BOOL; {access Read Only}   // 1=P_PIDE_Only AOI has been modified to include Autotune par. on PIDE block
   OCmd_ResetAckAll : BOOL;   // Operator Command to Reset all Alarms and latched Shed conditions
   OCmd_Reset : BOOL;   // Operator Command to Reset all Alarms requiring Reset
   MCmd_Check : BOOL;   // Maintenance Command to Check (not bypass) all Interlocks
   MCmd_Bypass : BOOL;   // Maintenance Command to Bypass all Bypassable Interlocks
   OCmd_SPRampStop : BOOL;   // Operator Command to stop SP ramping
   OCmd_SPRampStart : BOOL;   // Operator Command to initiate SP ramping
   OCmd_NormLM : BOOL;   // Operator Command to select Normal Loop Mode (see Cfg_NormLM)
   OCmd_Man : BOOL;   // Operator Command to select Manual control
   OCmd_Auto : BOOL;   // Operator Command to select Automatic control
   OCmd_Casc : BOOL;   // Operator Command to select Cascade / Ratio control
   OSet_CV : REAL;   // Operator Setting for Controlled Variable (loop Manual) (CVEU)
   OSet_SPRampT : REAL;   // Operator Setting for Setpoint Ramp Time (to reach target, for ramp wizard) (sec)
   OSet_SPTarget : REAL;   // Operator Setting for Setpoint Ramp Target (endpoint, for ramp wizard) (PVEU)
   OSet_SPRoCLimDec : REAL;   // Operator Setting for Setpoint Rate of Change Limit Decreasing (PVEU/sec)
   OSet_SPRoCLimInc : REAL;   // Operator Setting for Setpoint Rate of Change Limit Increasing (PVEU/sec)
   OSet_SP : REAL;   // Operator Setting for Setpoint (loop Auto) (PVEU)
   OSet_Ratio : REAL := 1.0;   // Operator Setting for Ratio (loop CasRat and Ratio enabled) (unitless)
   Wrk_ExtHas : SINT; {access None}   // External owns: .0=LM, .1=CV, .2=SP, .3=Ratio
   Wrk_ProgHas : SINT; {access None}   // Program owns: .0=LM, .1=CV, .2=SP, .3=Ratio
   Wrk_OperHas : SINT; {access None}   // Operator owns: .0=LM, .1=CV, .2=SP, .3=Ratio
   ORdy_SPRampT : BOOL; {access Read Only}   // 1=Ready for OSet_SPRampT (enables data entry field)
   ORdy_SPTarget : BOOL; {access Read Only}   // 1=Ready for OSet_SPTarget (enables data entry field)
   ORdy_CV : BOOL; {access Read Only}   // 1=Ready for OSet_CV (enables data entry field)
   ORdy_SP : BOOL; {access Read Only}   // 1=Ready for OSet_SP (enables data entry field)
   ORdy_Ratio : BOOL; {access Read Only}   // 1=Ready for OSet_Ratio (enables data entry field)
   ORdy_ResetAckAll : BOOL; {access Read Only}   // 1=At least one Alarm or latched Shed condition requires Reset or Ack
   ORdy_Reset : BOOL; {access Read Only}   // 1=Ready for OCmd_Reset (enables HMI button)
   MRdy_Check : BOOL; {access Read Only}   // 1=Ready for MCmd_Check (enables HMI button)
   MRdy_Bypass : BOOL; {access Read Only}   // 1=Ready for MCmd_Bypass (enables HMI button)
   ORdy_SPRampStop : BOOL; {access Read Only}   // 1=Ready for OCmd_RampStop (enables HMI button)
   ORdy_SPRampStart : BOOL; {access Read Only}   // 1=Ready for OCmd_RampSP (enables HMI button)
   ORdy_NormLM : BOOL; {access Read Only}   // 1=Ready for OCmd_NormLM (enables HMI button)
   ORdy_Man : BOOL; {access Read Only}   // 1=Ready for OCmd_Man (enables HMI button)
   ORdy_Auto : BOOL; {access Read Only}   // 1=Ready for OCmd_Auto (enables HMI button)
   ORdy_Casc : BOOL; {access Read Only}   // 1=Ready for OCmd_Casc (enables HMI button)
   Wrk_RealChkDINT : DINT; {access None}   // REAL bit pattern as a DINT for F.P. exception checking
   Wrk_PVInfNaN : BOOL; {access None}   // 1=PV is infinite or not a number
   Wrk_CascSPInfNaN : BOOL; {access None}   // Cascade Setpoint is Infinite or Not a Number
   Wrk_LoLoDev : BOOL; {access None}   // Internal flag: Low-Low Deviation Status
   Wrk_HiHiDev : BOOL; {access None}   // Internal flag: High-High Deviation Status
   Wrk_LoDev : BOOL; {access None}   // Internal flag: Low Deviation Status
   Wrk_HiDev : BOOL; {access None}   // Internal flag: High Deviation Status
   Wrk_FirstPIDCalc : BOOL; {access None}   // PID Not Skipped ONS store
   Wrk_HoldAtPV : BOOL; {access None}   // Shed SP equal to current PV One-Shot Store
   ORdy_SPRoCLimInc : BOOL; {access Read Only}   // 1=Ready for OSet_SPRoCLimInc (enables data entry field)
   ORdy_SPRoCLimDec : BOOL; {access Read Only}   // 1=Ready for OSet_SPRoCLimDec (enables data entry field)
   Wrk_Init : BOOL; {access None}   // 1=AOI has been initialized
   Wrk_SPRoCLimDec : REAL; {access None}   // Actual SP Rate of Change Limit Decreasing
   Wrk_SPRoCLimInc : REAL; {access None}   // Actual SP Rate of Change Limit Increasing
   Wrk_SPRampBusy : BOOL; {access None}   // 1=SP Ramp Wizard ramp is in progress
   Wrk_RatioClamped : BOOL; {access None}   // Buffer for building Sts_RatioClamped
END_VAR

ROUTINE EnableInFalse   (* ladder *)
// Disabled is asserted, output is set to configured Interlock CV, alarms are disabled
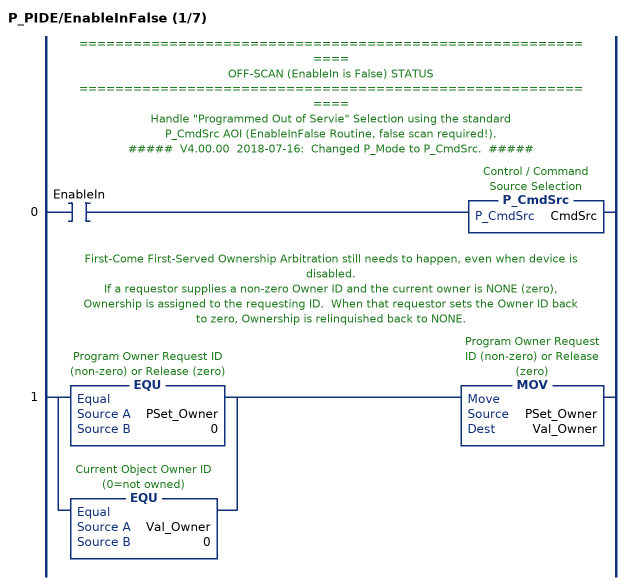
   // ============================================================
   // OFF-SCAN (EnableIn is False) STATUS
   // ============================================================
   // Handle "Programmed Out of Servie" Selection using the standard
   // P_CmdSrc AOI (EnableInFalse Routine, false scan required!).
   // #####  V4.00.00  2018-07-16:  Changed P_Mode to P_CmdSrc.  #####
   0: XIC(EnableIn)P_CmdSrc(CmdSrc);
   // First-Come First-Served Ownership Arbitration still needs to happen, even when device is disabled.
   // If a requestor supplies a non-zero Owner ID and the current owner is NONE (zero),
   // Ownership is assigned to the requesting ID.  When that requestor sets the Owner ID back
   // to zero, Ownership is relinquished back to NONE.
   1: [EQU(PSet_Owner,0) ,EQU(Val_Owner,0) ]MOV(PSet_Owner,Val_Owner);
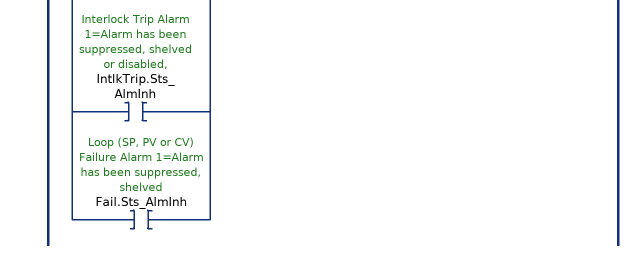
   // If the device is OFF-SCAN (rung is false or EnableIn is false in FBD),
   // then show the alarms as "Parent object out of service".
   // Show the overall acknowledgement status.
   // #####  V4.00.00  2018-07-16:  Changed P_Mode to P_CmdSrc, added Out of Service.  #####
   2: [OTL(HiHiDev.Inp_OoS) P_Alarm(HiHiDev) ,OTL(HiDev.Inp_OoS) P_Alarm(HiDev) ,OTL(LoDev.Inp_OoS) P_Alarm(LoDev) ,OTL(LoLoDev.Inp_OoS) P_Alarm(LoLoDev) ,OTL(IntlkTrip.Inp_OoS) P_Alarm(IntlkTrip) ,OTL(Fail.Inp_OoS) P_Alarm(Fail) ,CLR(Val_Notify) CLR(Val_NotifyAll) ,[XIC(HiHiDev.Val_Notify.0) ,XIC(HiDev.Val_Notify.0) ,XIC(LoDev.Val_Notify.0) ,XIC(LoLoDev.Val_Notify.0) ,XIC(IntlkTrip.Val_Notify.0) ,XIC(Fail.Val_Notify.0) ] OTL(Val_Notify.0) OTL(Val_NotifyAll.0) ,[XIC(HiHiDev.Sts_AlmInh) ,XIC(HiDev.Sts_AlmInh) ,XIC(LoDev.Sts_AlmInh) ,XIC(LoLoDev.Sts_AlmInh) ,XIC(IntlkTrip.Sts_AlmInh) ,XIC(Fail.Sts_AlmInh) ] OTE(Sts_AlmInh) ];
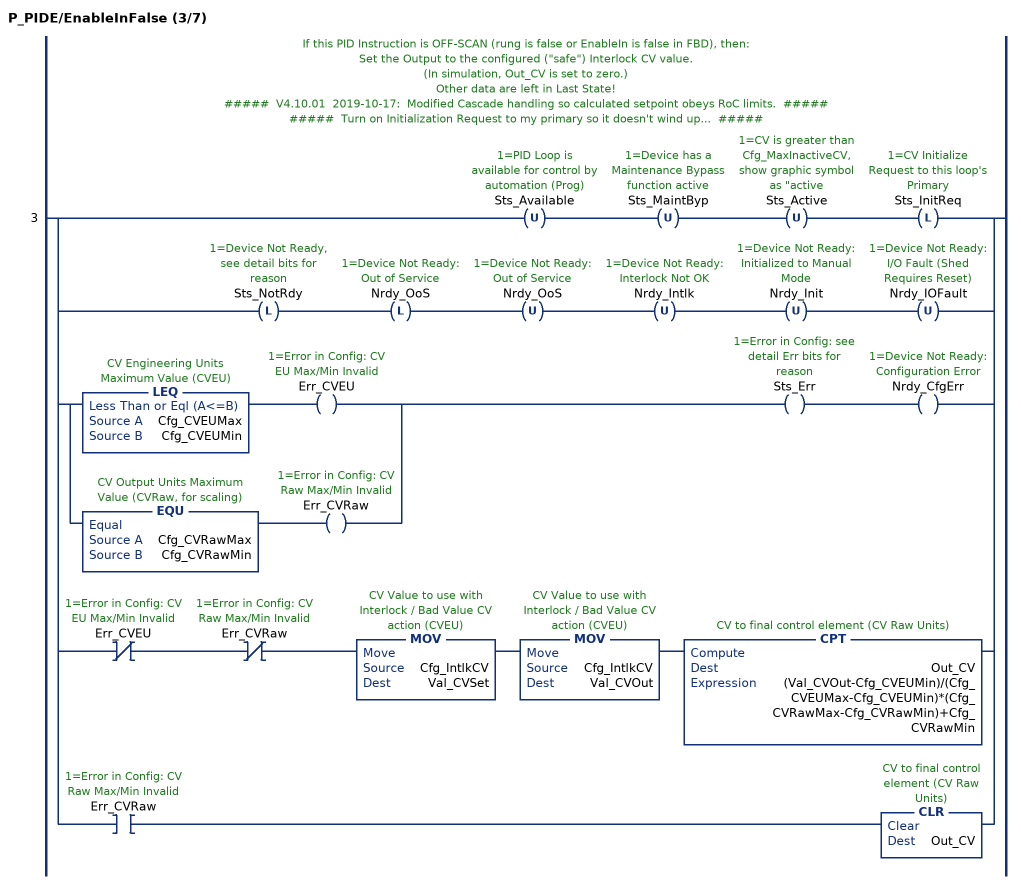
   // If this PID Instruction is OFF-SCAN (rung is false or EnableIn is false in FBD), then:
   // Set the Output to the configured ("safe") Interlock CV value.
   // (In simulation, Out_CV is set to zero.)
   // Other data are left in Last State!
   // #####  V4.10.01  2019-10-17:  Modified Cascade handling so calculated setpoint obeys RoC limits.  #####
   // #####  Turn on Initialization Request to my primary so it doesn't wind up...  #####
   3: [OTU(Sts_Available) OTU(Sts_MaintByp) OTU(Sts_Active) OTL(Sts_InitReq) ,OTL(Sts_NotRdy) OTL(Nrdy_OoS) OTU(Nrdy_OoS) OTU(Nrdy_Intlk) OTU(Nrdy_Init) OTU(Nrdy_IOFault) ,[LEQ(Cfg_CVEUMax,Cfg_CVEUMin) OTE(Err_CVEU) ,EQU(Cfg_CVRawMax,Cfg_CVRawMin) OTE(Err_CVRaw) ] OTE(Sts_Err) OTE(Nrdy_CfgErr) ,XIO(Err_CVEU) XIO(Err_CVRaw) MOV(Cfg_IntlkCV,Val_CVSet) MOV(Cfg_IntlkCV,Val_CVOut) CPT(Out_CV,(Val_CVOut-Cfg_CVEUMin)/(Cfg_CVEUMax-Cfg_CVEUMin)*(Cfg_CVRawMax-Cfg_CVRawMin)+Cfg_CVRawMin) ,XIC(Err_CVRaw) CLR(Out_CV) ];
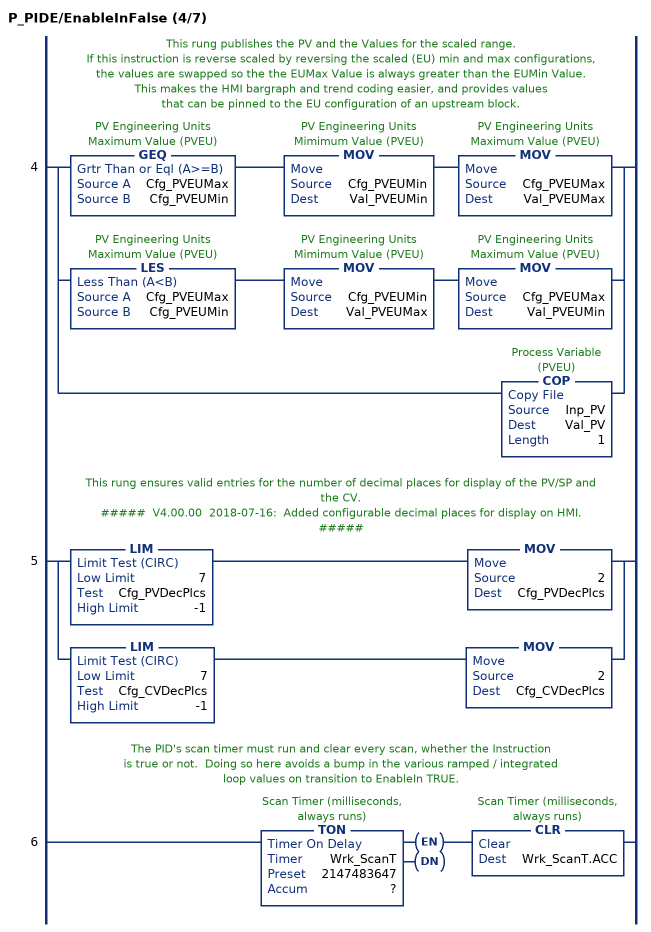
   // This rung publishes the PV and the Values for the scaled range.
   // If this instruction is reverse scaled by reversing the scaled (EU) min and max configurations,
   // the values are swapped so the the EUMax Value is always greater than the EUMin Value.
   // This makes the HMI bargraph and trend coding easier, and provides values
   // that can be pinned to the EU configuration of an upstream block.
   4: [GEQ(Cfg_PVEUMax,Cfg_PVEUMin) MOV(Cfg_PVEUMin,Val_PVEUMin) MOV(Cfg_PVEUMax,Val_PVEUMax) ,LES(Cfg_PVEUMax,Cfg_PVEUMin) MOV(Cfg_PVEUMin,Val_PVEUMax) MOV(Cfg_PVEUMax,Val_PVEUMin) ,COP(Inp_PV,Val_PV,1) ];
   // This rung ensures valid entries for the number of decimal places for display of the PV/SP and the CV.
   // #####  V4.00.00  2018-07-16:  Added configurable decimal places for display on HMI.  #####
   5: [LIM(7,Cfg_PVDecPlcs,-1) MOV(2,Cfg_PVDecPlcs) ,LIM(7,Cfg_CVDecPlcs,-1) MOV(2,Cfg_CVDecPlcs) ];
   // The PID's scan timer must run and clear every scan, whether the Instruction
   // is true or not.  Doing so here avoids a bump in the various ramped / integrated
   // loop values on transition to EnableIn TRUE.
   6: TON(Wrk_ScanT,?,?)CLR(Wrk_ScanT.ACC);
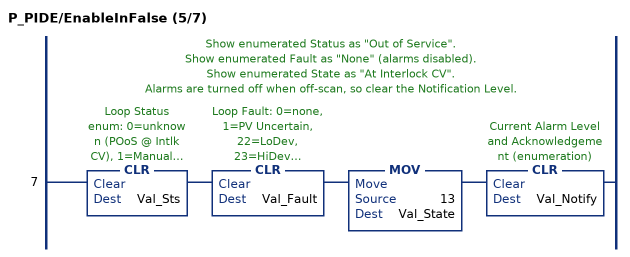
   // Show enumerated Status as "Out of Service".
   // Show enumerated Fault as "None" (alarms disabled).
   // Show enumerated State as "At Interlock CV".
   // Alarms are turned off when off-scan, so clear the Notification Level.
   7: CLR(Val_Sts)CLR(Val_Fault)MOV(13,Val_State)CLR(Val_Notify);
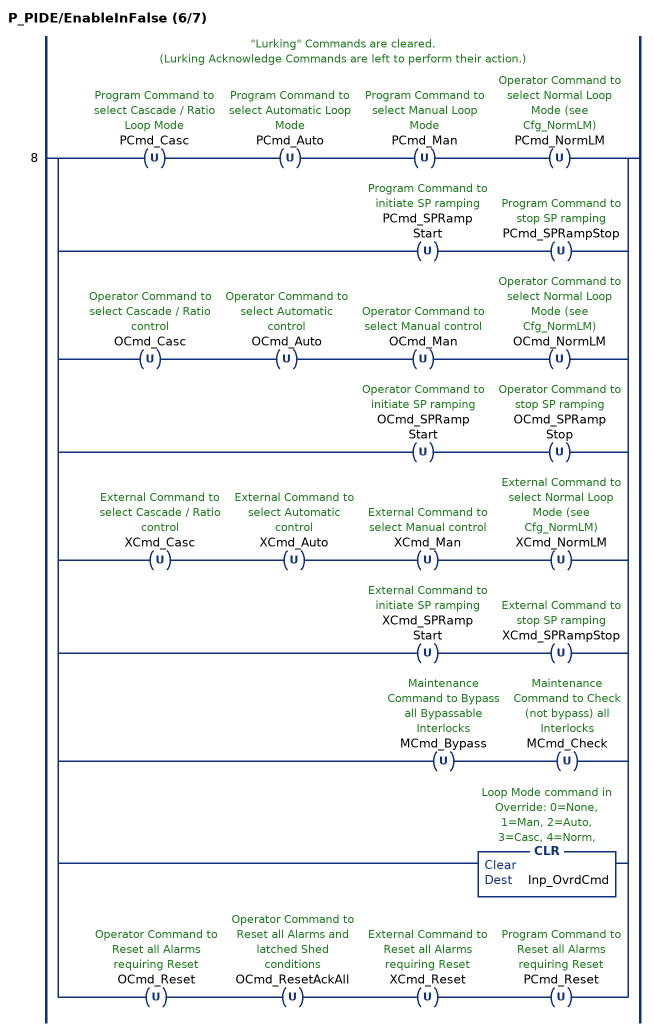
   // "Lurking" Commands are cleared.
   // (Lurking Acknowledge Commands are left to perform their action.)
   8: [OTU(PCmd_Casc) OTU(PCmd_Auto) OTU(PCmd_Man) OTU(PCmd_NormLM) ,OTU(PCmd_SPRampStart) OTU(PCmd_SPRampStop) ,OTU(OCmd_Casc) OTU(OCmd_Auto) OTU(OCmd_Man) OTU(OCmd_NormLM) ,OTU(OCmd_SPRampStart) OTU(OCmd_SPRampStop) ,OTU(XCmd_Casc) OTU(XCmd_Auto) OTU(XCmd_Man) OTU(XCmd_NormLM) ,OTU(XCmd_SPRampStart) OTU(XCmd_SPRampStop) ,OTU(MCmd_Bypass) OTU(MCmd_Check) ,CLR(Inp_OvrdCmd) ,OTU(OCmd_Reset) OTU(OCmd_ResetAckAll) OTU(XCmd_Reset) OTU(PCmd_Reset) ];
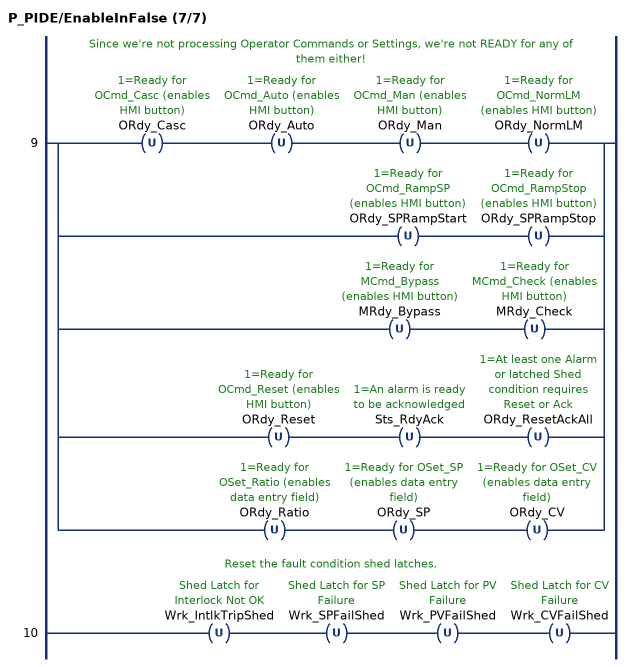
   // Since we're not processing Operator Commands or Settings, we're not READY for any of them either!
   9: [OTU(ORdy_Casc) OTU(ORdy_Auto) OTU(ORdy_Man) OTU(ORdy_NormLM) ,OTU(ORdy_SPRampStart) OTU(ORdy_SPRampStop) ,OTU(MRdy_Bypass) OTU(MRdy_Check) ,OTU(ORdy_Reset) OTU(Sts_RdyAck) OTU(ORdy_ResetAckAll) ,OTU(ORdy_Ratio) OTU(ORdy_SP) OTU(ORdy_CV) ];
   // Reset the fault condition shed latches.
   10: OTU(Wrk_IntlkTripShed)OTU(Wrk_SPFailShed)OTU(Wrk_PVFailShed)OTU(Wrk_CVFailShed);
END_ROUTINE
